// TIA Portal V20 export
// export: Created 2025-12-01T14:57:39.8501249Z, ExportSetting None, DisplayName Totally Integrated Automation Portal, DisplayVersion V20 Update 3, DisplayName TIA Portal Openness, DisplayVersion V20 Update 3, DisplayName TIA Portal Version Control Interface, DisplayVersion V20 Update 3, DisplayName STEP 7 Professional, DisplayVersion V20 Update 3, DisplayName STEP 7 Safety, DisplayVersion V20 Update 2, DisplayName WinCC Basic/Comfort/Advanced, DisplayVersion V20 Update 3, DisplayName WinCC Professional, DisplayVersion V20 Update 3, DisplayName WinCC Unified, DisplayVersion V20 Update 3
FUNCTION_BLOCK "FB371_DesApiladorDeCajasPlastico"   // FB371, LAD
TITLE = DesApilador de Cajas de Plastico
{ S7_Optimized_Access := 'FALSE' }
AUTHOR : MAQUINA
NAME : 20160211
VERSION : 3.2
// Dani Palacios: Modificación octubre 2017 para poder desabilitar la maquina con un bit (por ejemplo en la puesta a punto si no esta montada o en el simulador)
// La modificación esta sin probar y es todo lo relativo a la variable MaquinaDesHabilitada
// (bloqueo evolución desde etapa 0, bloqueo activación salidas en etapa 0 , fin vi sin mirar detectores y activación posición de reposo sin mirar detectores y variabkles de fin de movimiento).
// ES RESPONSABILIDAD DEL QUE DESABILITA LA MAQUINA QUE ESTA ESTE EN UNA POSICION QUE PERMITA EL MOVIMIENTO DE LAS CARGAS A TRAVES DE ELLA
// stored: AutoNumber false, SetENOAutomatically false
   VAR_INPUT
      Maquina : UInt;   // Numero de Maquina (Mesa)
      Error_Tx : Bool;   // Error en el Tx
      EnTension : Bool;   // Existe Tension en la Mesa
      NodoNoPresente : Bool;   // Nodo No Presente >>> Var. LENZE de Elevacion
      ByteInicial : Int;   // Byte Inicial >>> Var. LENZE de Elevacion
      MAQx_DesHabilitada : Bool;   // Config MAQ. >>> DesHabilitada
      MAQx_SinCentrador : Bool;   // Config MAQ. >>> No Activar Centrador
      MAQx_ActivarEspera : Bool;   // Config MAQ. >>> Sin Espera en Etapas
      TermicoFreno_ELEV : Bool;   // Termico del Freno de la Elevacion
      pHsMx_PresCarga : Bool;   // pHs de Presencia de Carga en la Maquina
      pHsMx_1 : Bool;   // pHs de la Mesa - Pos 1 de Av
      pHsMx_2 : Bool;   // pHs de la Mesa - Pos 2 de Av
      pHsMx_CrtSalida : Bool;   // pHs Control de Salida de Seguridad
      pHs_Referencia : Bool;   // pHs de Referencia >>> Var. LENZE de Elevacion
      EM_Up : Bool;   // Emergencia Arriba >>> Var. LENZE de Elevacion
      EM_Down : Bool;   // Emergencia Abajo >>> Var. LENZE de Elevacion
      CF1CF2_Cerrado : Bool;   // Centradores 1 y 2 Cerrados
      CF3CF4_Cerrado : Bool;   // Centradores 3 y 4 Cerrados
      CF5CF6_Cerrado : Bool;   // Centradores 5 y 6 Cerrados
      CF1CF2_Abierto : Bool;   // Centradores 1 y 2 Abiertos
      CF3CF4_Abierto : Bool;   // Centradores 3 y 4 Abiertos
      CF5CF6_Abierto : Bool;   // Centradores 5 y 6 Abiertos
      CM1CM2_Cerrado : Bool;   // Garras 1 y 2 Cerradas
      CM3CM4_Cerrado : Bool;   // Garras 3 y 4 Cerradas
      CM5CM6_Cerrado : Bool;   // Garras 5 y 6 Cerradas
      CM7CM8_Cerrado : Bool;   // Garras 7 y 8 Cerradas
      CM9CM10_Cerrado : Bool;   // Garras 9 y 10 Cerradas
      CM1CM2_Abierto : Bool;   // Garras 1 y 2 Abiertas
      CM3CM4_Abierto : Bool;   // Garras 3 y 4 Abiertas
      CM5CM6_Abierto : Bool;   // Garras 5 y 6 Abiertas
      CM7CM8_Abierto : Bool;   // Garras 7 y 8 Abiertas
      CM9CM10_Abierto : Bool;   // Garras 9 y 10 Abiertas
      GF1GF2_Cerrado : Bool;   // Guias superiores 1 y 2 Cerradas
      GF3GF4_Cerrado : Bool;   // Guias superiores 3 y 4 Cerradas
      GF1GF2_Abierto : Bool;   // Guias superiores 1 y 2 Abiertas
      GF3GF4_Abierto : Bool;   // Guias superiores 3 y 4 Abiertas
      EnMov_Centradores : Bool;   // Centradores >>> En Movimiento
      EnMov_Garras : Bool;   // Garras >>> En Movimiento
      EnMov_Guias : Bool;   // Guias >>> En Movimiento
      SubirManual : Bool;   // Subir en Manual >>> Var. LENZE de Elevacion
      BajarManual : Bool;   // Bajar en Manual >>> Var. LENZE de Elevacion
      AutoManual : Bool;   // Posicionar en Manual (Para realizar Test de Posicion)
      Homing : Bool;   // Homing >>> Var. LENZE de Elevacion
      DesApilador_FinSalida : Bool;   // Fin Salida >>> Interlock Mesa
      ActivarGuias : Bool;   // Activar las Guias Superiores (Por altura de la Pila)
      V_TOut_MovVertical : Int := 15000;   // TimeOut del Movimiento Vertical
      V_TOut_Centradores : Int := 5000;   // TimeOut de los Centradores
      V_TOut_Garras : Int := 5000;   // TimeOut de las Garras
      V_TOut_Guias : Int := 5000;   // TimeOut de las Guias Superiores
   END_VAR
   VAR_OUTPUT
      DesApilador_EnReposo : Bool;   // En Reposo >>> Interlock Maquina
      DesApilador_PermisoSalida : Bool;   // Permiso de Salida >>> Interlock Maquina
   END_VAR
   VAR
      PosicionActual : Int;   // Var. LENZE de Elevacion >>> Posicion Actual
      ErrorSubjet : Word;   // Var LENZE de Elevacion
      ErrorID : Word;   // Var LENZE de Elevacion
      PosicionManual : UInt;   // Posicion para el Test Manual
      PosicionInicial : UInt;   // TRACKING >>> Posicion Inicial de la Orden de DesApilar Cajas
      PosicionFinal : UInt;   // TRACKING >>> Posicion Final de la Orden de DesApilar Cajas
      TipoAmarre : UInt;   // TRACKING >>> Tipo de Amarre de las Garras de la Orden de DesApilar Cajas
      OrdenDesApilar : Bool;   // TRACKING >>> Orden de DesApilar Cajas
      Fin_OrdenDesApilar : Bool;   // TRACKING >>> Fin de la Orden de DesApilar Cajas
      Caja_TipoEuroPool : Bool;   // TRACKING >>> Caja de tipo EuroPool
      Caja_DosPequenas : Bool;   // TRACKING >>> La Fila es de Dos Cajas Pequeñas
      Caja_UnaPequena : Bool;   // TRACKING >>> La Fila es de Una Caja Pequeña
      Caja_Grande : Bool;   // TRACKING >>> La Fila es de Una Caja Grande
      EnPila_UnicaFila : Bool;   // TRACKING >>> La Pila es de Una Unica Fila
      Reset_ET00 : Bool;
      Reset_ET01 : Bool;
      DesApil_ET00 : Bool;
      DesApil_ET01 : Bool;
      DesApil_ET02 : Bool;
      DesApil_ET03 : Bool;
      DesApil_ET04 : Bool;
      DesApil_ET05 : Bool;
      DesApil_ET06 : Bool;
      DesApil_ET07 : Bool;
      DesApil_ET08 : Bool;
      PosicionIntermedia : UInt;   // AUXILIAR >>> Posicion Internedia de la Orden a Mover el Elevacion
      Posicion_OrdenMover : UInt;   // AUXILIAR >>> Posicion de la Orden a Mover el Elevacion
      OrdenMover : Bool;   // AUXILIAR >>> Orden de Mover el Elevacion
      Fin_OrdenMover : Bool;   // AUXILIAR >>> Orden de Mover el Elevacion
      MemoPosicionOK : Bool;   // AUXILIAR >>> Memoria de Posicion OK
      Carga_PosicionInicial : Bool;   // CARGA >>> Posicion Incial del DesApilado de Cajas
      Carga_PosicionIntermedia : Bool;   // CARGA >>> Posicion Intermedia del DesApilado de Cajas
      Carga_PosicionFinal : Bool;   // CARGA >>> Posicion Final del DesApilado de Cajas
      Carga_PosicionManual : Bool;   // CARGA >>> Posicion Manual de la Orden de Test
      ErrorVariador : Bool;   // AUXILIAR >>> Error del Variador
      ReferenciaOK : Bool;   // AUXILIAR >>> Referencia OK del Variador
      MemoHomingAuto : Bool;   // AUXILIAR >>> Memoria del Homing Automatico del Variador
      TIM_EsperaMover { S7_SetPoint := 'True'} : TON_TIME;   // TIM de Espera de Activar Orden al Var de LENZE (200ms)
      TIM_EsperaET02 { S7_SetPoint := 'True'} : TON_TIME;   // TIM de Espera para Activar ET02 (100ms)
      TIM_EsperaET04 { S7_SetPoint := 'True'} : TON_TIME;   // TIM de Espera para Activar ET04 (100ms)
      TMP_EnTension { S7_SetPoint := 'True'} : "FB910_CNT_UHS";
      TOut_MovVertical { S7_SetPoint := 'True'} : "FB910_CNT_UHS";   // TimeOut del Movimiento Vertical
      TOut_Centradores { S7_SetPoint := 'True'} : "FB910_CNT_UHS";   // TimeOut de los Centradores
      TOut_Garras { S7_SetPoint := 'True'} : "FB910_CNT_UHS";   // TimeOut de las Garras
      TOut_Guias { S7_SetPoint := 'True'} : "FB910_CNT_UHS";   // TimeOut de las Guias Superiores
      MA_Cerrar_CF1CF2 : Bool;   // ???
      MA_Cerrar_CF3CF4 : Bool;   // ???
      MA_Cerrar_CF5CF6 : Bool;   // ???
      MA_Abrir_CF1CF2 : Bool;   // ???
      MA_Abrir_CF3CF4 : Bool;   // ???
      MA_Abrir_CF5CF6 : Bool;   // ???
      MA_Cerrar_CM1CM2 : Bool;   // ???
      MA_Cerrar_CM3CM4 : Bool;   // ???
      MA_Cerrar_CM5CM6 : Bool;   // ???
      MA_Cerrar_CM7CM8 : Bool;   // ???
      MA_Cerrar_CM9CM10 : Bool;   // ???
      MA_Abrir_CM1CM2 : Bool;   // ???
      MA_Abrir_CM3CM4 : Bool;   // ???
      MA_Abrir_CM5CM6 : Bool;   // ???
      MA_Abrir_CM7CM8 : Bool;   // ???
      MA_Abrir_CM9CM10 : Bool;   // ???
      MA_Cerrar_GF1GF2 : Bool;   // ???
      MA_Cerrar_GF3GF4 : Bool;   // ???
      MA_Abrir_GF1GF2 : Bool;   // ???
      MA_Abrir_GF3GF4 : Bool;   // ???
   END_VAR
   VAR_TEMP
      EstadoZona : "EstadoZona";   // Estado de Zona de la Mesa
      EstadoMAQ : "EstadoMaquina_DesApiladorDeCajasPlastico";   // Estado del Vehiculo Inteliguente de la Maquina
      MAQx_AutoHoming : Bool;   // Config >>> Var. LENZE con Auto Homing
      MAQx_EncoderIncremental : Bool;   // Config >>> Var. LENZE con Encoder Incremental
      MAQx_ActivarAutoManual : Bool;   // Config >>> Activacion para el Test de posicionamiento manual
      CentradoresCerrados : Bool;   // AUXILIAR >>> Cerrados los Centradores
      CentradoresAbiertos : Bool;   // AUXILIAR >>> Abiertos los Centradores
      GarrasCerradas : Bool;   // AUXILIAR >>> Cerradas las Garras
      GarrasAbiertas : Bool;   // AUXILIAR >>> Abiertas las Garras
      GuiasCerradas : Bool;   // AUXILIAR >>> Cerradas las Guias Superiores
      GuiasAbiertas : Bool;   // AUXILIAR >>> Abiertas las Guias Superiores
      MA_CerrarCentradores : Bool;   // AUXILIAR >>> Cerrar los Centradores
      MA_AbrirCentradores : Bool;   // AUXILIAR >>> Abrir los Centradores
      MA_CerrarGarras : Bool;   // AUXILIAR >>> Cerrar las Garras
      MA_AbrirGarras : Bool;   // AUXILIAR >>> Abrir las Garras
      MA_CerrarGuias : Bool;   // AUXILIAR >>> Cerrar las Guias Superiores
      MA_AbrirGuias : Bool;   // AUXILIAR >>> Abrir las Guias Superiores
      AuxEstados : Bool;
   END_VAR
BEGIN

REGION Network 1: Configuraciones Especiales - Config >>> Var. LENZE de Elevacion
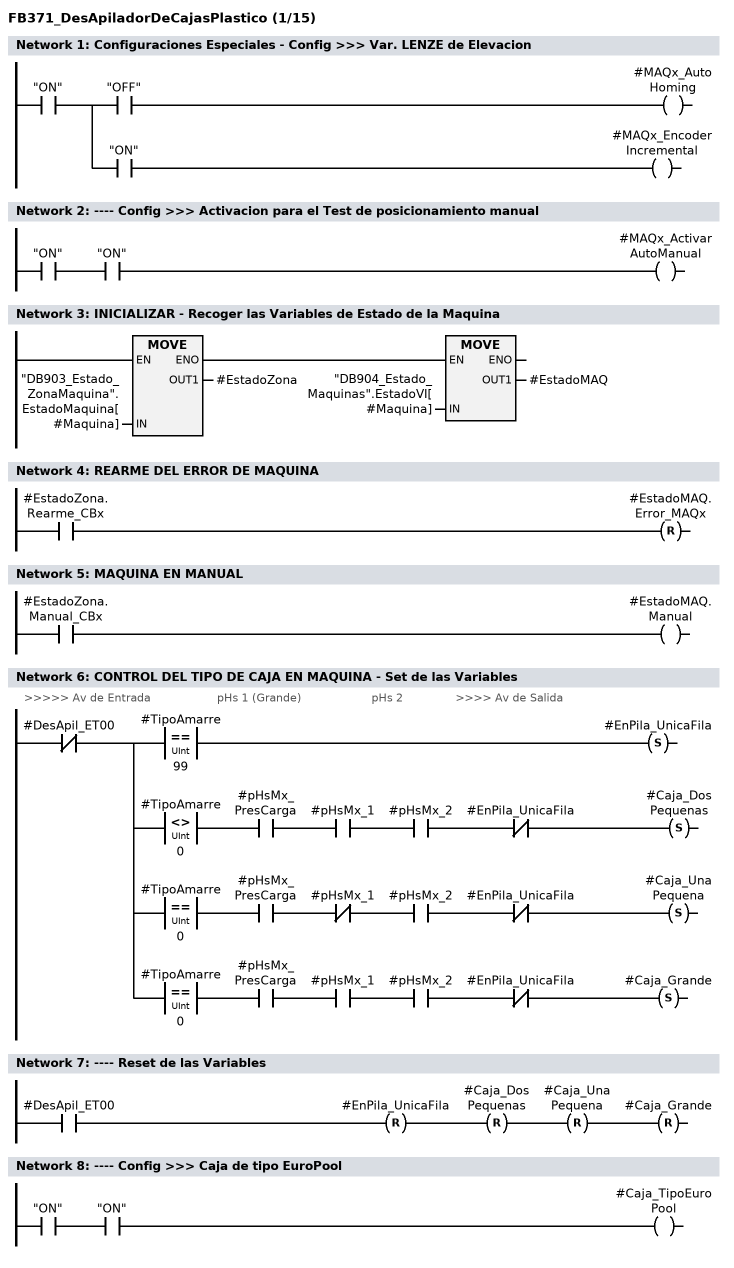
   RUNG wire#powerrail
      Contact( "ON" )
      wire#w1
      Contact( "OFF" )
      Coil( #MAQx_AutoHoming )
   END_RUNG
   RUNG wire#w1
      Contact( "ON" )
      Coil( #MAQx_EncoderIncremental )
   END_RUNG
   // the same network as SCL:
   #MAQx_AutoHoming := "ON" AND "OFF";
   #MAQx_EncoderIncremental := "ON" AND "ON";
END_REGION

REGION Network 2: ---- Config >>> Activacion para el Test de posicionamiento manual
   RUNG wire#powerrail
      Contact( "ON" )
      Contact( "ON" )
      Coil( #MAQx_ActivarAutoManual )
   END_RUNG
   // the same network as SCL:
   #MAQx_ActivarAutoManual := "ON" AND "ON";
END_REGION

REGION Network 3: INICIALIZAR - Recoger las Variables de Estado de la Maquina
   RUNG wire#powerrail
      Move(in := "DB903_Estado_ZonaMaquina".EstadoMaquina[#Maquina], out1 => #EstadoZona)
      Move(in := "DB904_Estado_Maquinas".EstadoVI[#Maquina], out1 => #EstadoMAQ)
   END_RUNG
   // the same network as SCL:
   #EstadoZona := "DB903_Estado_ZonaMaquina".EstadoMaquina[#Maquina];
   #EstadoMAQ := "DB904_Estado_Maquinas".EstadoVI[#Maquina];
END_REGION

REGION Network 4: REARME DEL ERROR DE MAQUINA
   RUNG wire#powerrail
      Contact( #EstadoZona.Rearme_CBx )
      R_Coil( #EstadoMAQ.Error_MAQx )
   END_RUNG
   // the same network as SCL:
   IF #EstadoZona.Rearme_CBx THEN #EstadoMAQ.Error_MAQx := FALSE; END_IF;
END_REGION

REGION Network 5: MAQUINA EN MANUAL
   RUNG wire#powerrail
      Contact( #EstadoZona.Manual_CBx )
      Coil( #EstadoMAQ.Manual )
   END_RUNG
   // the same network as SCL:
   #EstadoMAQ.Manual := #EstadoZona.Manual_CBx;
END_REGION

REGION Network 6: CONTROL DEL TIPO DE CAJA EN MAQUINA - Set de las Variables
   // >>>>> Av de Entrada                   pHs 1 (Grande)                    pHs 2               >>>> Av de Salida
   RUNG wire#powerrail
      I_Contact( #DesApil_ET00 )
      wire#w1
      { S7_Templates := "SrcType := UInt" } EQ_Contact(in1 := #TipoAmarre, in2 := 99)
      S_Coil( #EnPila_UnicaFila )
   END_RUNG
   RUNG wire#w1
      { S7_Templates := "SrcType := UInt" } NE_Contact(in1 := #TipoAmarre, in2 := 0)
      Contact( #pHsMx_PresCarga )
      Contact( #pHsMx_1 )
      Contact( #pHsMx_2 )
      I_Contact( #EnPila_UnicaFila )
      S_Coil( #Caja_DosPequenas )
   END_RUNG
   RUNG wire#w1
      { S7_Templates := "SrcType := UInt" } EQ_Contact(in1 := #TipoAmarre, in2 := 0)
      Contact( #pHsMx_PresCarga )
      I_Contact( #pHsMx_1 )
      Contact( #pHsMx_2 )
      I_Contact( #EnPila_UnicaFila )
      S_Coil( #Caja_UnaPequena )
   END_RUNG
   RUNG wire#w1
      { S7_Templates := "SrcType := UInt" } EQ_Contact(in1 := #TipoAmarre, in2 := 0)
      Contact( #pHsMx_PresCarga )
      Contact( #pHsMx_1 )
      Contact( #pHsMx_2 )
      I_Contact( #EnPila_UnicaFila )
      S_Coil( #Caja_Grande )
   END_RUNG
   // the same network as SCL:
   IF NOT #DesApil_ET00 AND (#TipoAmarre = 99) THEN #EnPila_UnicaFila := TRUE; END_IF;
   IF NOT #DesApil_ET00 AND (#TipoAmarre <> 0) AND #pHsMx_PresCarga AND #pHsMx_1 AND #pHsMx_2 AND NOT #EnPila_UnicaFila THEN
       #Caja_DosPequenas := TRUE;
   END_IF;
   IF NOT #DesApil_ET00 AND (#TipoAmarre = 0) AND #pHsMx_PresCarga AND NOT #pHsMx_1 AND #pHsMx_2 AND NOT #EnPila_UnicaFila THEN
       #Caja_UnaPequena := TRUE;
   END_IF;
   IF NOT #DesApil_ET00 AND (#TipoAmarre = 0) AND #pHsMx_PresCarga AND #pHsMx_1 AND #pHsMx_2 AND NOT #EnPila_UnicaFila THEN
       #Caja_Grande := TRUE;
   END_IF;
END_REGION

REGION Network 7: ---- Reset de las Variables
   RUNG wire#powerrail
      Contact( #DesApil_ET00 )
      R_Coil( #EnPila_UnicaFila )
      R_Coil( #Caja_DosPequenas )
      R_Coil( #Caja_UnaPequena )
      R_Coil( #Caja_Grande )
   END_RUNG
   // the same network as SCL:
   IF #DesApil_ET00 THEN
       #EnPila_UnicaFila := FALSE;
       #Caja_DosPequenas := FALSE;
       #Caja_UnaPequena := FALSE;
       #Caja_Grande := FALSE;
   END_IF;
END_REGION

REGION Network 8: ---- Config >>> Caja de tipo EuroPool
   RUNG wire#powerrail
      Contact( "ON" )
      Contact( "ON" )
      Coil( #Caja_TipoEuroPool )
   END_RUNG
   // the same network as SCL:
   #Caja_TipoEuroPool := "ON" AND "ON";
END_REGION

REGION Network 9: VARIABLES AUXILIARES - Control de Centradores - Cerrados
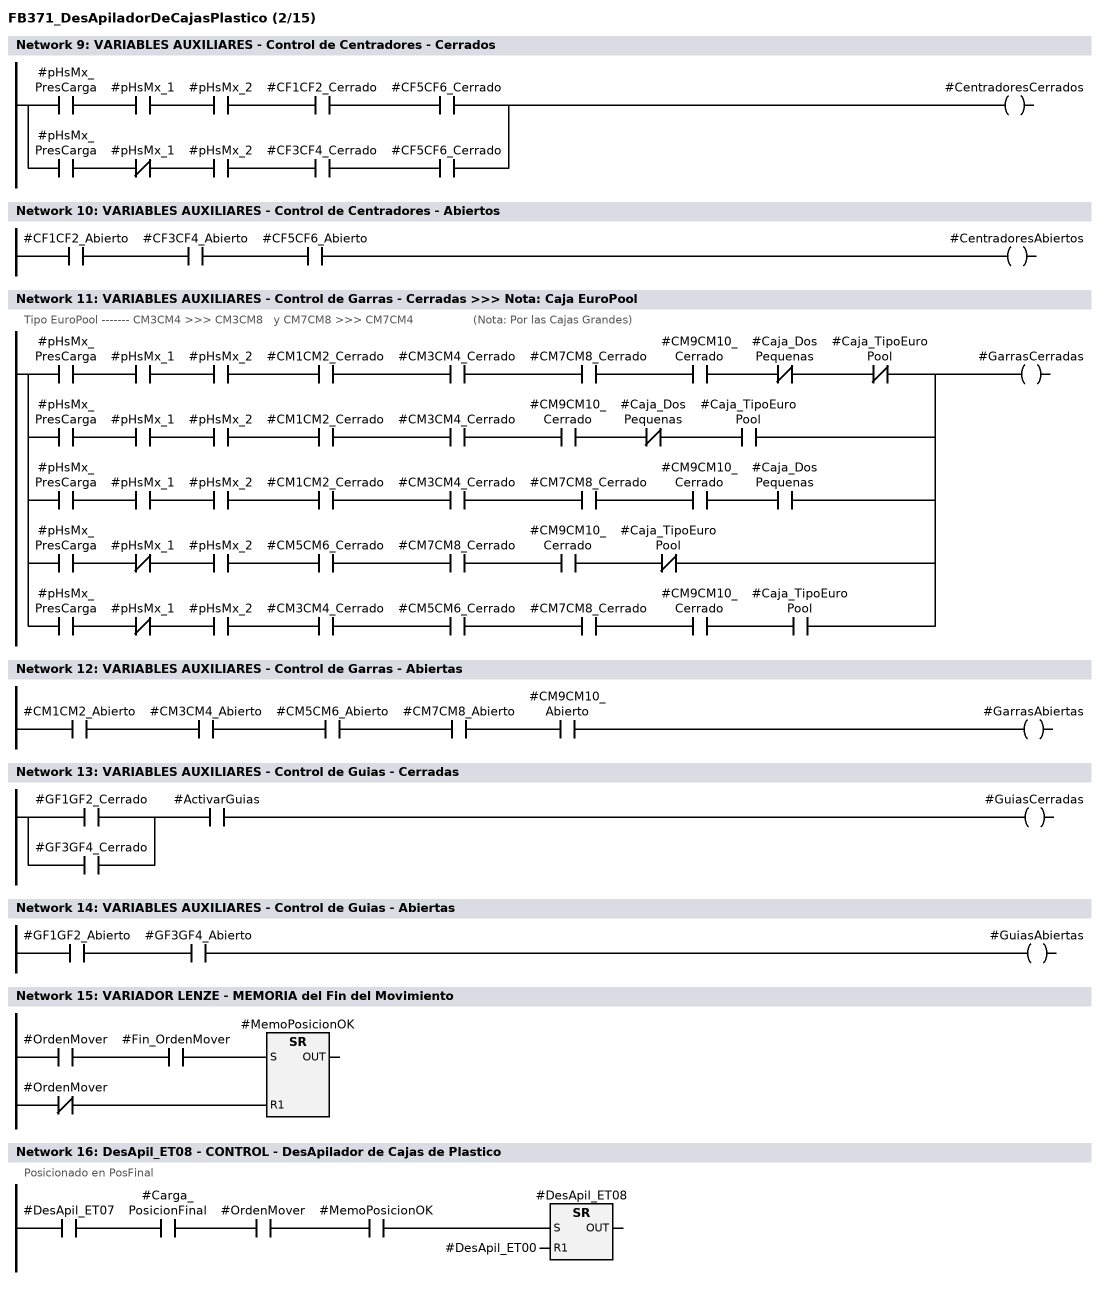
   RUNG wire#powerrail
      Contact( #pHsMx_PresCarga )
      Contact( #pHsMx_1 )
      Contact( #pHsMx_2 )
      Contact( #CF1CF2_Cerrado )
      Contact( #CF5CF6_Cerrado )
      wire#w1
      Coil( #CentradoresCerrados )
   END_RUNG
   RUNG wire#powerrail
      Contact( #pHsMx_PresCarga )
      I_Contact( #pHsMx_1 )
      Contact( #pHsMx_2 )
      Contact( #CF3CF4_Cerrado )
      Contact( #CF5CF6_Cerrado )
   END_RUNG wire#w1
   // the same network as SCL:
   #CentradoresCerrados := (#pHsMx_PresCarga AND #pHsMx_1 AND #pHsMx_2 AND #CF1CF2_Cerrado AND #CF5CF6_Cerrado) OR (#pHsMx_PresCarga AND NOT #pHsMx_1 AND #pHsMx_2 AND #CF3CF4_Cerrado AND #CF5CF6_Cerrado);
END_REGION

REGION Network 10: VARIABLES AUXILIARES - Control de Centradores - Abiertos
   RUNG wire#powerrail
      Contact( #CF1CF2_Abierto )
      Contact( #CF3CF4_Abierto )
      Contact( #CF5CF6_Abierto )
      Coil( #CentradoresAbiertos )
   END_RUNG
   // the same network as SCL:
   #CentradoresAbiertos := #CF1CF2_Abierto AND #CF3CF4_Abierto AND #CF5CF6_Abierto;
END_REGION

REGION Network 11: VARIABLES AUXILIARES - Control de Garras - Cerradas >>> Nota: Caja EuroPool
   // Tipo EuroPool ------- CM3CM4 >>> CM3CM8   y CM7CM8 >>> CM7CM4                 (Nota: Por las Cajas Grandes)
   RUNG wire#powerrail
      Contact( #pHsMx_PresCarga )
      Contact( #pHsMx_1 )
      Contact( #pHsMx_2 )
      Contact( #CM1CM2_Cerrado )
      Contact( #CM3CM4_Cerrado )
      Contact( #CM7CM8_Cerrado )
      Contact( #CM9CM10_Cerrado )
      I_Contact( #Caja_DosPequenas )
      I_Contact( #Caja_TipoEuroPool )
      wire#w1
      Coil( #GarrasCerradas )
   END_RUNG
   RUNG wire#powerrail
      Contact( #pHsMx_PresCarga )
      Contact( #pHsMx_1 )
      Contact( #pHsMx_2 )
      Contact( #CM1CM2_Cerrado )
      Contact( #CM3CM4_Cerrado )
      Contact( #CM9CM10_Cerrado )
      I_Contact( #Caja_DosPequenas )
      Contact( #Caja_TipoEuroPool )
   END_RUNG wire#w1
   RUNG wire#powerrail
      Contact( #pHsMx_PresCarga )
      Contact( #pHsMx_1 )
      Contact( #pHsMx_2 )
      Contact( #CM1CM2_Cerrado )
      Contact( #CM3CM4_Cerrado )
      Contact( #CM7CM8_Cerrado )
      Contact( #CM9CM10_Cerrado )
      Contact( #Caja_DosPequenas )
   END_RUNG wire#w1
   RUNG wire#powerrail
      Contact( #pHsMx_PresCarga )
      I_Contact( #pHsMx_1 )
      Contact( #pHsMx_2 )
      Contact( #CM5CM6_Cerrado )
      Contact( #CM7CM8_Cerrado )
      Contact( #CM9CM10_Cerrado )
      I_Contact( #Caja_TipoEuroPool )
   END_RUNG wire#w1
   RUNG wire#powerrail
      Contact( #pHsMx_PresCarga )
      I_Contact( #pHsMx_1 )
      Contact( #pHsMx_2 )
      Contact( #CM3CM4_Cerrado )
      Contact( #CM5CM6_Cerrado )
      Contact( #CM7CM8_Cerrado )
      Contact( #CM9CM10_Cerrado )
      Contact( #Caja_TipoEuroPool )
   END_RUNG wire#w1
   // the same network as SCL:
   #GarrasCerradas := (#pHsMx_PresCarga AND #pHsMx_1 AND #pHsMx_2 AND #CM1CM2_Cerrado AND #CM3CM4_Cerrado AND #CM7CM8_Cerrado AND #CM9CM10_Cerrado AND NOT #Caja_DosPequenas AND NOT #Caja_TipoEuroPool) OR (#pHsMx_PresCarga AND #pHsMx_1 AND #pHsMx_2 AND #CM1CM2_Cerrado AND #CM3CM4_Cerrado AND #CM9CM10_Cerrado AND NOT #Caja_DosPequenas AND #Caja_TipoEuroPool) OR (#pHsMx_PresCarga AND #pHsMx_1 AND #pHsMx_2 AND #CM1CM2_Cerrado AND #CM3CM4_Cerrado AND #CM7CM8_Cerrado AND #CM9CM10_Cerrado AND #Caja_DosPequenas) OR (#pHsMx_PresCarga AND NOT #pHsMx_1 AND #pHsMx_2 AND #CM5CM6_Cerrado AND #CM7CM8_Cerrado AND #CM9CM10_Cerrado AND NOT #Caja_TipoEuroPool) OR (#pHsMx_PresCarga AND NOT #pHsMx_1 AND #pHsMx_2 AND #CM3CM4_Cerrado AND #CM5CM6_Cerrado AND #CM7CM8_Cerrado AND #CM9CM10_Cerrado AND #Caja_TipoEuroPool);
END_REGION

REGION Network 12: VARIABLES AUXILIARES - Control de Garras - Abiertas
   RUNG wire#powerrail
      Contact( #CM1CM2_Abierto )
      Contact( #CM3CM4_Abierto )
      Contact( #CM5CM6_Abierto )
      Contact( #CM7CM8_Abierto )
      Contact( #CM9CM10_Abierto )
      Coil( #GarrasAbiertas )
   END_RUNG
   // the same network as SCL:
   #GarrasAbiertas := #CM1CM2_Abierto AND #CM3CM4_Abierto AND #CM5CM6_Abierto AND #CM7CM8_Abierto AND #CM9CM10_Abierto;
END_REGION

REGION Network 13: VARIABLES AUXILIARES - Control de Guias - Cerradas
   RUNG wire#powerrail
      Contact( #GF1GF2_Cerrado )
      wire#w1
      Contact( #ActivarGuias )
      Coil( #GuiasCerradas )
   END_RUNG
   RUNG wire#powerrail
      Contact( #GF3GF4_Cerrado )
   END_RUNG wire#w1
   // the same network as SCL:
   #GuiasCerradas := (#GF1GF2_Cerrado OR #GF3GF4_Cerrado) AND #ActivarGuias;
END_REGION

REGION Network 14: VARIABLES AUXILIARES - Control de Guias - Abiertas
   RUNG wire#powerrail
      Contact( #GF1GF2_Abierto )
      Contact( #GF3GF4_Abierto )
      Coil( #GuiasAbiertas )
   END_RUNG
   // the same network as SCL:
   #GuiasAbiertas := #GF1GF2_Abierto AND #GF3GF4_Abierto;
END_REGION

REGION Network 15: VARIADOR LENZE - MEMORIA del Fin del Movimiento
   RUNG wire#powerrail
      Contact( #OrdenMover )
      Contact( #Fin_OrdenMover )
      S_SR(operand := #MemoPosicionOK, r1 := wire#w1)
   END_RUNG
   RUNG wire#powerrail
      I_Contact( #OrdenMover )
   END_RUNG wire#w1
   // the same network as SCL:
   IF #OrdenMover AND #Fin_OrdenMover THEN
       #MemoPosicionOK := TRUE;   // SR flip-flop
   END_IF;
   IF NOT #OrdenMover THEN #MemoPosicionOK := FALSE; END_IF;
END_REGION

REGION Network 16: DesApil_ET08 - CONTROL - DesApilador de Cajas de Plastico
   // Posicionado en PosFinal
   RUNG wire#powerrail
      Contact( #DesApil_ET07 )
      Contact( #Carga_PosicionFinal )
      Contact( #OrdenMover )
      Contact( #MemoPosicionOK )
      S_SR(operand := #DesApil_ET08, r1 := #DesApil_ET00)
   END_RUNG
   // the same network as SCL:
   IF #DesApil_ET07 AND #Carga_PosicionFinal AND #OrdenMover AND #MemoPosicionOK THEN
       #DesApil_ET08 := TRUE;   // SR flip-flop
   END_IF;
   IF #DesApil_ET00 THEN #DesApil_ET08 := FALSE; END_IF;
END_REGION

REGION Network 17: DesApil_ET07
   // A Salido la Caja
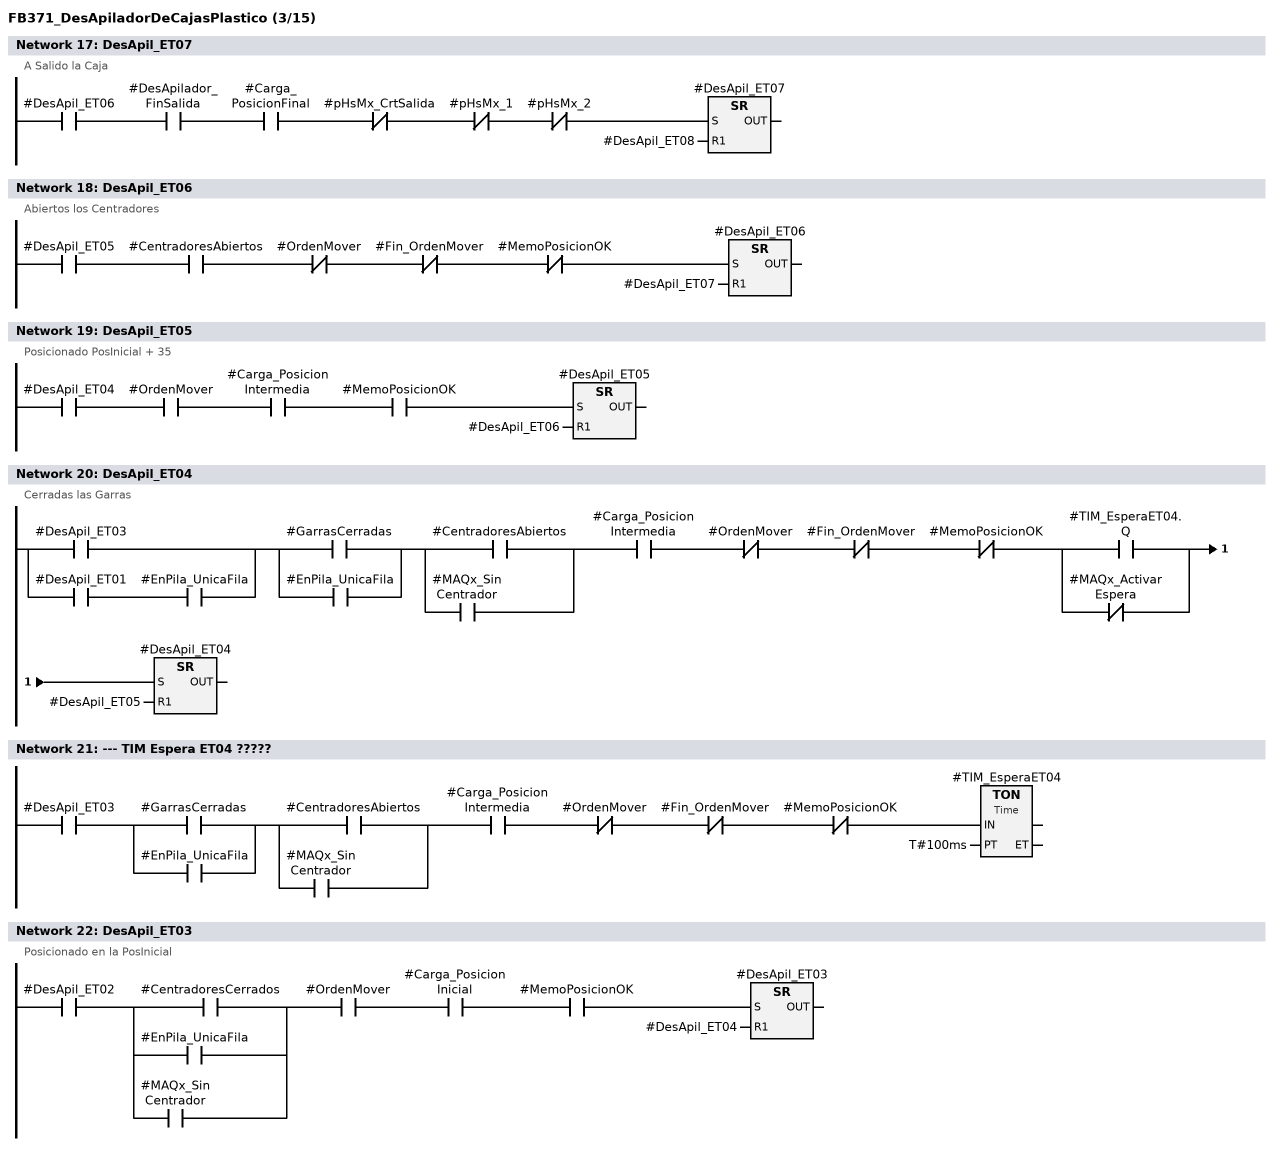
   RUNG wire#powerrail
      Contact( #DesApil_ET06 )
      Contact( #DesApilador_FinSalida )
      Contact( #Carga_PosicionFinal )
      I_Contact( #pHsMx_CrtSalida )
      I_Contact( #pHsMx_1 )
      I_Contact( #pHsMx_2 )
      S_SR(operand := #DesApil_ET07, r1 := #DesApil_ET08)
   END_RUNG
   // the same network as SCL:
   IF #DesApil_ET06 AND #DesApilador_FinSalida AND #Carga_PosicionFinal AND NOT #pHsMx_CrtSalida AND NOT #pHsMx_1 AND NOT #pHsMx_2 THEN
       #DesApil_ET07 := TRUE;   // SR flip-flop
   END_IF;
   IF #DesApil_ET08 THEN #DesApil_ET07 := FALSE; END_IF;
END_REGION

REGION Network 18: DesApil_ET06
   // Abiertos los Centradores
   RUNG wire#powerrail
      Contact( #DesApil_ET05 )
      Contact( #CentradoresAbiertos )
      I_Contact( #OrdenMover )
      I_Contact( #Fin_OrdenMover )
      I_Contact( #MemoPosicionOK )
      S_SR(operand := #DesApil_ET06, r1 := #DesApil_ET07)
   END_RUNG
   // the same network as SCL:
   IF #DesApil_ET05 AND #CentradoresAbiertos AND NOT #OrdenMover AND NOT #Fin_OrdenMover AND NOT #MemoPosicionOK THEN
       #DesApil_ET06 := TRUE;   // SR flip-flop
   END_IF;
   IF #DesApil_ET07 THEN #DesApil_ET06 := FALSE; END_IF;
END_REGION

REGION Network 19: DesApil_ET05
   // Posicionado PosInicial + 35
   RUNG wire#powerrail
      Contact( #DesApil_ET04 )
      Contact( #OrdenMover )
      Contact( #Carga_PosicionIntermedia )
      Contact( #MemoPosicionOK )
      S_SR(operand := #DesApil_ET05, r1 := #DesApil_ET06)
   END_RUNG
   // the same network as SCL:
   IF #DesApil_ET04 AND #OrdenMover AND #Carga_PosicionIntermedia AND #MemoPosicionOK THEN
       #DesApil_ET05 := TRUE;   // SR flip-flop
   END_IF;
   IF #DesApil_ET06 THEN #DesApil_ET05 := FALSE; END_IF;
END_REGION

REGION Network 20: DesApil_ET04
   // Cerradas las Garras
   RUNG wire#powerrail
      Contact( #DesApil_ET03 )
      wire#w1
      Contact( #GarrasCerradas )
      wire#w2
      Contact( #CentradoresAbiertos )
      wire#w3
      Contact( #Carga_PosicionIntermedia )
      I_Contact( #OrdenMover )
      I_Contact( #Fin_OrdenMover )
      I_Contact( #MemoPosicionOK )
      wire#w4
      Contact( #TIM_EsperaET04.Q )
      wire#w5
      S_SR(operand := #DesApil_ET04, r1 := #DesApil_ET05)
   END_RUNG
   RUNG wire#powerrail
      Contact( #DesApil_ET01 )
      Contact( #EnPila_UnicaFila )
   END_RUNG wire#w1
   RUNG wire#w1
      Contact( #EnPila_UnicaFila )
   END_RUNG wire#w2
   RUNG wire#w2
      Contact( #MAQx_SinCentrador )
   END_RUNG wire#w3
   RUNG wire#w4
      I_Contact( #MAQx_ActivarEspera )
   END_RUNG wire#w5
   // the same network as SCL:
   IF (#DesApil_ET03 OR (#DesApil_ET01 AND #EnPila_UnicaFila)) AND (#GarrasCerradas OR #EnPila_UnicaFila) AND (#CentradoresAbiertos OR #MAQx_SinCentrador) AND #Carga_PosicionIntermedia AND NOT #OrdenMover AND NOT #Fin_OrdenMover AND NOT #MemoPosicionOK AND (#TIM_EsperaET04.Q OR NOT #MAQx_ActivarEspera) THEN
       #DesApil_ET04 := TRUE;   // SR flip-flop
   END_IF;
   IF #DesApil_ET05 THEN #DesApil_ET04 := FALSE; END_IF;
END_REGION

REGION Network 21: --- TIM Espera ET04 ?????
   RUNG wire#powerrail
      Contact( #DesApil_ET03 )
      wire#w1
      Contact( #GarrasCerradas )
      wire#w2
      Contact( #CentradoresAbiertos )
      wire#w3
      Contact( #Carga_PosicionIntermedia )
      I_Contact( #OrdenMover )
      I_Contact( #Fin_OrdenMover )
      I_Contact( #MemoPosicionOK )
      { S7_Templates := "time_type := Time" } #TIM_EsperaET04.TON(pt := T#100ms, et =>)
   END_RUNG
   RUNG wire#w1
      Contact( #EnPila_UnicaFila )
   END_RUNG wire#w2
   RUNG wire#w2
      Contact( #MAQx_SinCentrador )
   END_RUNG wire#w3
   // the same network as SCL:
   #TIM_EsperaET04(IN := #DesApil_ET03 AND (#GarrasCerradas OR #EnPila_UnicaFila) AND (#CentradoresAbiertos OR #MAQx_SinCentrador) AND #Carga_PosicionIntermedia AND NOT #OrdenMover AND NOT #Fin_OrdenMover AND NOT #MemoPosicionOK,   // TON
                   PT := T#100ms);
END_REGION

REGION Network 22: DesApil_ET03
   // Posicionado en la PosInicial
   RUNG wire#powerrail
      Contact( #DesApil_ET02 )
      wire#w1
      Contact( #CentradoresCerrados )
      wire#w2
      Contact( #OrdenMover )
      Contact( #Carga_PosicionInicial )
      Contact( #MemoPosicionOK )
      S_SR(operand := #DesApil_ET03, r1 := #DesApil_ET04)
   END_RUNG
   RUNG wire#w1
      Contact( #EnPila_UnicaFila )
   END_RUNG wire#w2
   RUNG wire#w1
      Contact( #MAQx_SinCentrador )
   END_RUNG wire#w2
   // the same network as SCL:
   IF #DesApil_ET02 AND (#CentradoresCerrados OR #EnPila_UnicaFila OR #MAQx_SinCentrador) AND #OrdenMover AND #Carga_PosicionInicial AND #MemoPosicionOK THEN
       #DesApil_ET03 := TRUE;   // SR flip-flop
   END_IF;
   IF #DesApil_ET04 THEN #DesApil_ET03 := FALSE; END_IF;
END_REGION

REGION Network 23: DesApil_ET02
   // Cerrados los Centradores
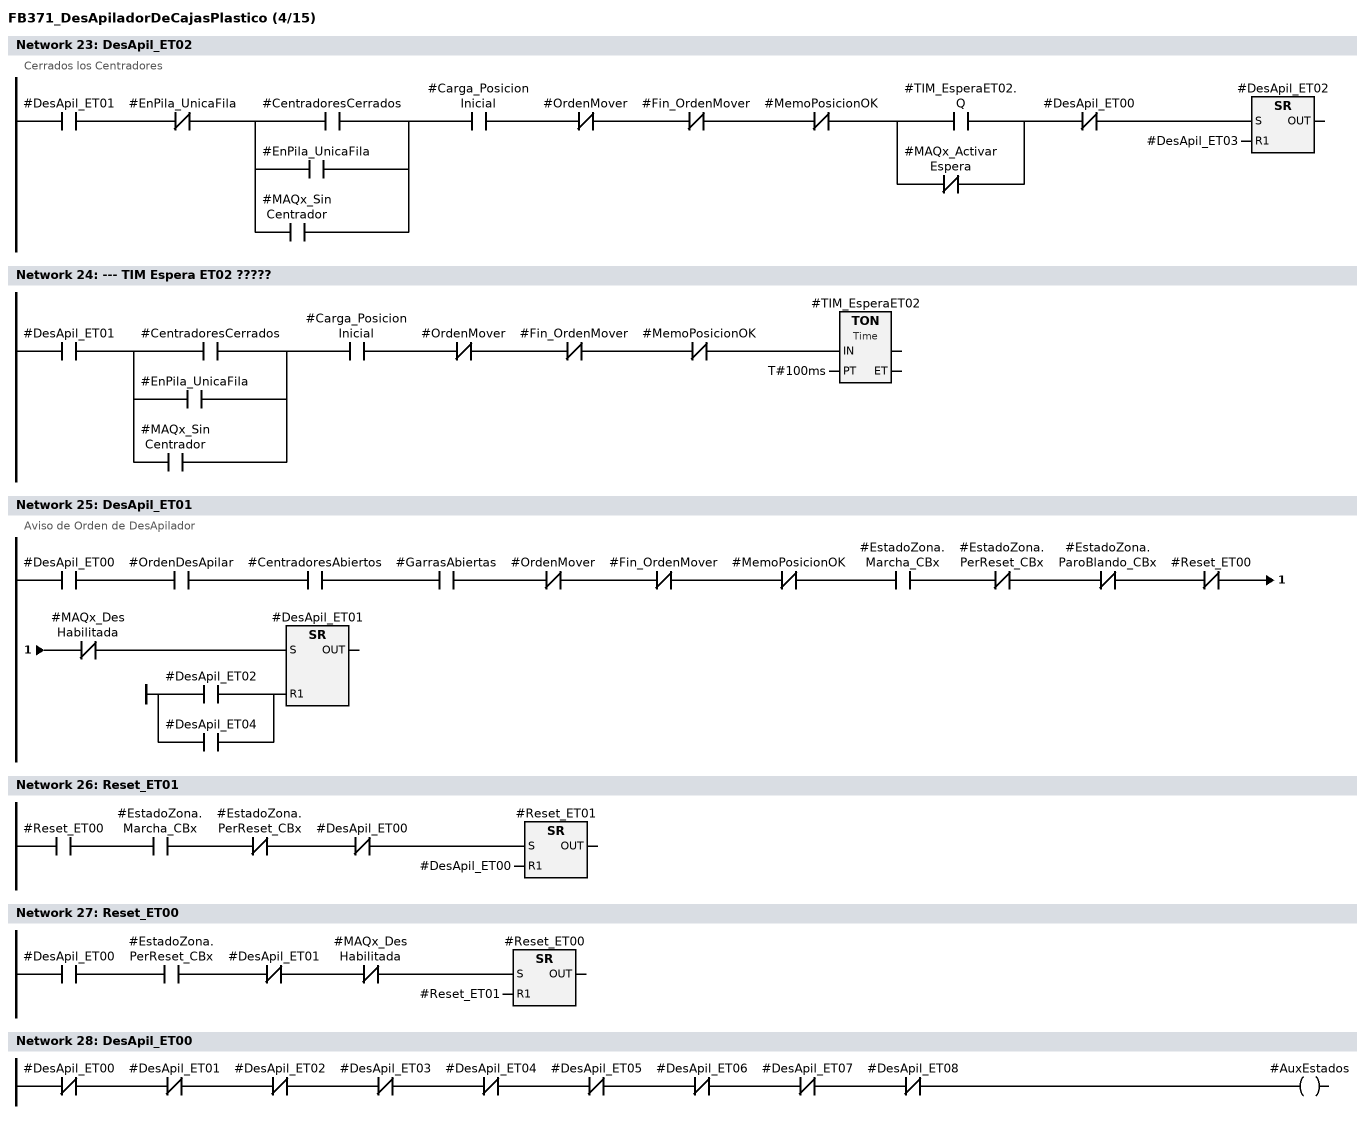
   RUNG wire#powerrail
      Contact( #DesApil_ET01 )
      I_Contact( #EnPila_UnicaFila )
      wire#w1
      Contact( #CentradoresCerrados )
      wire#w2
      Contact( #Carga_PosicionInicial )
      I_Contact( #OrdenMover )
      I_Contact( #Fin_OrdenMover )
      I_Contact( #MemoPosicionOK )
      wire#w3
      Contact( #TIM_EsperaET02.Q )
      wire#w4
      I_Contact( #DesApil_ET00 )
      S_SR(operand := #DesApil_ET02, r1 := #DesApil_ET03)
   END_RUNG
   RUNG wire#w1
      Contact( #EnPila_UnicaFila )
   END_RUNG wire#w2
   RUNG wire#w1
      Contact( #MAQx_SinCentrador )
   END_RUNG wire#w2
   RUNG wire#w3
      I_Contact( #MAQx_ActivarEspera )
   END_RUNG wire#w4
   // the same network as SCL:
   IF #DesApil_ET01 AND NOT #EnPila_UnicaFila AND (#CentradoresCerrados OR #EnPila_UnicaFila OR #MAQx_SinCentrador) AND #Carga_PosicionInicial AND NOT #OrdenMover AND NOT #Fin_OrdenMover AND NOT #MemoPosicionOK AND (#TIM_EsperaET02.Q OR NOT #MAQx_ActivarEspera) AND NOT #DesApil_ET00 THEN
       #DesApil_ET02 := TRUE;   // SR flip-flop
   END_IF;
   IF #DesApil_ET03 THEN #DesApil_ET02 := FALSE; END_IF;
END_REGION

REGION Network 24: --- TIM Espera ET02 ?????
   RUNG wire#powerrail
      Contact( #DesApil_ET01 )
      wire#w1
      Contact( #CentradoresCerrados )
      wire#w2
      Contact( #Carga_PosicionInicial )
      I_Contact( #OrdenMover )
      I_Contact( #Fin_OrdenMover )
      I_Contact( #MemoPosicionOK )
      { S7_Templates := "time_type := Time" } #TIM_EsperaET02.TON(pt := T#100ms, et =>)
   END_RUNG
   RUNG wire#w1
      Contact( #EnPila_UnicaFila )
   END_RUNG wire#w2
   RUNG wire#w1
      Contact( #MAQx_SinCentrador )
   END_RUNG wire#w2
   // the same network as SCL:
   #TIM_EsperaET02(IN := #DesApil_ET01 AND (#CentradoresCerrados OR #EnPila_UnicaFila OR #MAQx_SinCentrador) AND #Carga_PosicionInicial AND NOT #OrdenMover AND NOT #Fin_OrdenMover AND NOT #MemoPosicionOK,   // TON
                   PT := T#100ms);
END_REGION

REGION Network 25: DesApil_ET01
   // Aviso de Orden de DesApilador
   RUNG wire#powerrail
      Contact( #DesApil_ET00 )
      Contact( #OrdenDesApilar )
      Contact( #CentradoresAbiertos )
      Contact( #GarrasAbiertas )
      I_Contact( #OrdenMover )
      I_Contact( #Fin_OrdenMover )
      I_Contact( #MemoPosicionOK )
      Contact( #EstadoZona.Marcha_CBx )
      I_Contact( #EstadoZona.PerReset_CBx )
      I_Contact( #EstadoZona.ParoBlando_CBx )
      I_Contact( #Reset_ET00 )
      I_Contact( #MAQx_DesHabilitada )
      S_SR(operand := #DesApil_ET01, r1 := wire#w1)
   END_RUNG
   RUNG wire#powerrail
      Contact( #DesApil_ET02 )
   END_RUNG wire#w1
   RUNG wire#powerrail
      Contact( #DesApil_ET04 )
   END_RUNG wire#w1
   // the same network as SCL:
   IF #DesApil_ET00 AND #OrdenDesApilar AND #CentradoresAbiertos AND #GarrasAbiertas AND NOT #OrdenMover AND NOT #Fin_OrdenMover AND NOT #MemoPosicionOK AND #EstadoZona.Marcha_CBx AND NOT #EstadoZona.PerReset_CBx AND NOT #EstadoZona.ParoBlando_CBx AND NOT #Reset_ET00 AND NOT #MAQx_DesHabilitada THEN
       #DesApil_ET01 := TRUE;   // SR flip-flop
   END_IF;
   IF #DesApil_ET02 OR #DesApil_ET04 THEN #DesApil_ET01 := FALSE; END_IF;
END_REGION

REGION Network 26: Reset_ET01
   RUNG wire#powerrail
      Contact( #Reset_ET00 )
      Contact( #EstadoZona.Marcha_CBx )
      I_Contact( #EstadoZona.PerReset_CBx )
      I_Contact( #DesApil_ET00 )
      S_SR(operand := #Reset_ET01, r1 := #DesApil_ET00)
   END_RUNG
   // the same network as SCL:
   IF #Reset_ET00 AND #EstadoZona.Marcha_CBx AND NOT #EstadoZona.PerReset_CBx AND NOT #DesApil_ET00 THEN
       #Reset_ET01 := TRUE;   // SR flip-flop
   END_IF;
   IF #DesApil_ET00 THEN #Reset_ET01 := FALSE; END_IF;
END_REGION

REGION Network 27: Reset_ET00
   RUNG wire#powerrail
      Contact( #DesApil_ET00 )
      Contact( #EstadoZona.PerReset_CBx )
      I_Contact( #DesApil_ET01 )
      I_Contact( #MAQx_DesHabilitada )
      S_SR(operand := #Reset_ET00, r1 := #Reset_ET01)
   END_RUNG
   // the same network as SCL:
   IF #DesApil_ET00 AND #EstadoZona.PerReset_CBx AND NOT #DesApil_ET01 AND NOT #MAQx_DesHabilitada THEN
       #Reset_ET00 := TRUE;   // SR flip-flop
   END_IF;
   IF #Reset_ET01 THEN #Reset_ET00 := FALSE; END_IF;
END_REGION

REGION Network 28: DesApil_ET00
   RUNG wire#powerrail
      I_Contact( #DesApil_ET00 )
      I_Contact( #DesApil_ET01 )
      I_Contact( #DesApil_ET02 )
      I_Contact( #DesApil_ET03 )
      I_Contact( #DesApil_ET04 )
      I_Contact( #DesApil_ET05 )
      I_Contact( #DesApil_ET06 )
      I_Contact( #DesApil_ET07 )
      I_Contact( #DesApil_ET08 )
      Coil( #AuxEstados )
   END_RUNG
   // the same network as SCL:
   #AuxEstados := NOT #DesApil_ET00 AND NOT #DesApil_ET01 AND NOT #DesApil_ET02 AND NOT #DesApil_ET03 AND NOT #DesApil_ET04 AND NOT #DesApil_ET05 AND NOT #DesApil_ET06 AND NOT #DesApil_ET07 AND NOT #DesApil_ET08;
END_REGION

REGION Network 29: ---
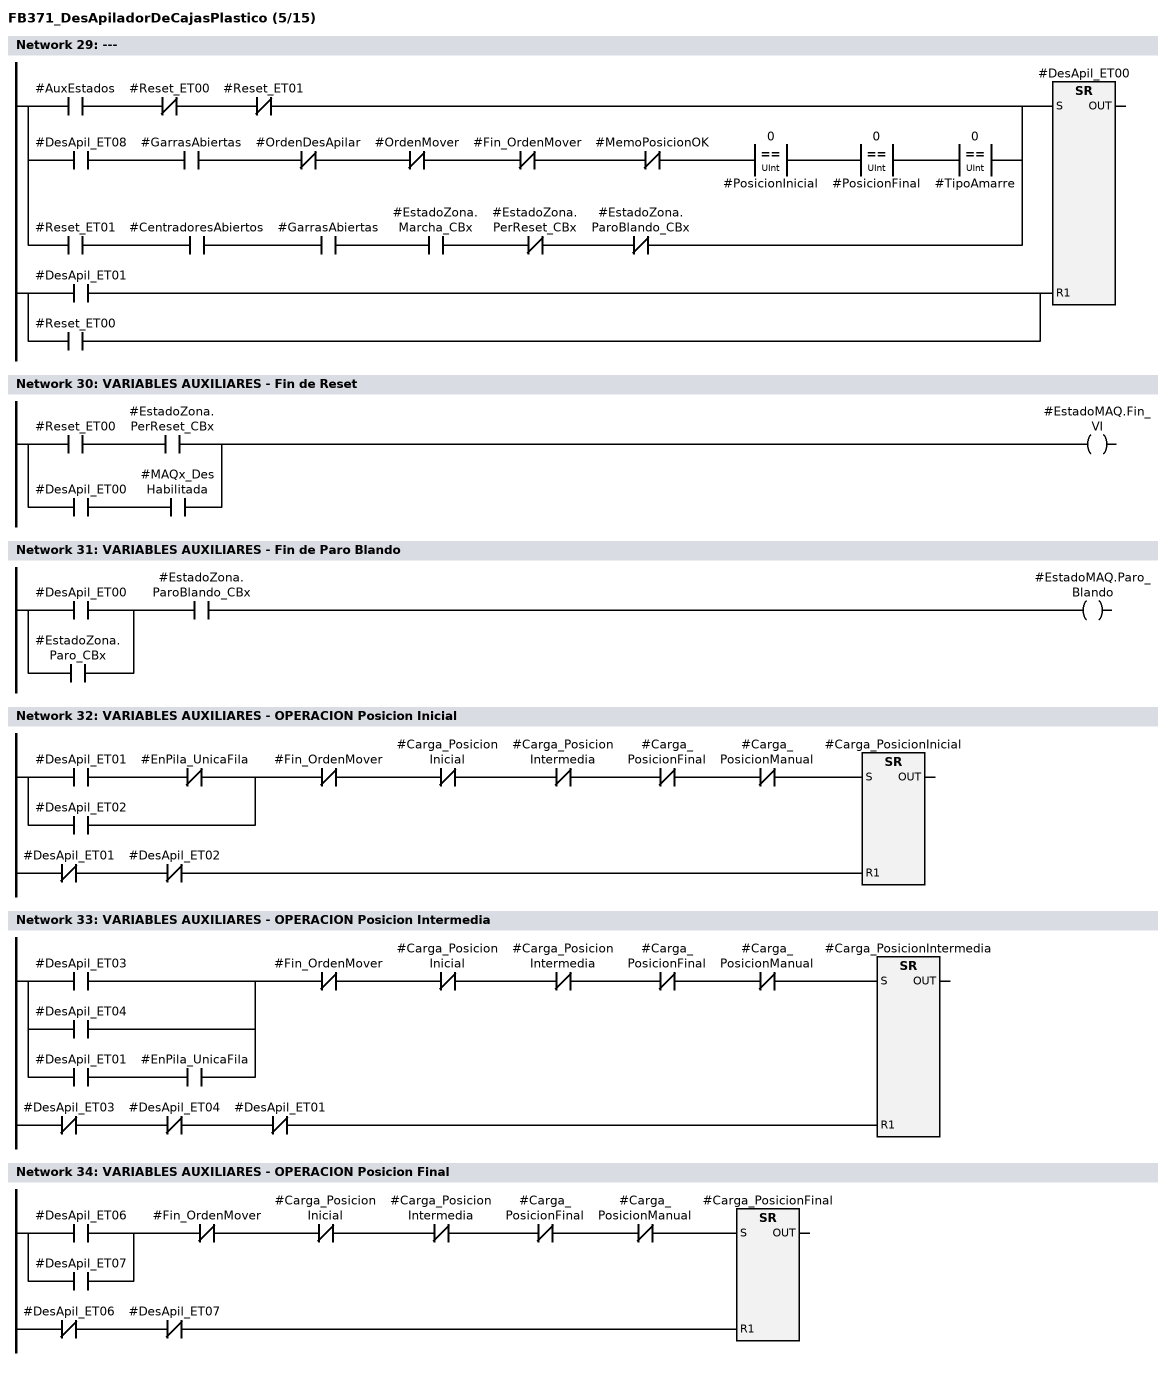
   RUNG wire#powerrail
      Contact( #AuxEstados )
      I_Contact( #Reset_ET00 )
      I_Contact( #Reset_ET01 )
      wire#w1
      S_SR(operand := #DesApil_ET00, r1 := wire#w2)
   END_RUNG
   RUNG wire#powerrail
      Contact( #DesApil_ET08 )
      Contact( #GarrasAbiertas )
      I_Contact( #OrdenDesApilar )
      I_Contact( #OrdenMover )
      I_Contact( #Fin_OrdenMover )
      I_Contact( #MemoPosicionOK )
      { S7_Templates := "SrcType := UInt" } EQ_Contact(in1 := 0, in2 := #PosicionInicial)
      { S7_Templates := "SrcType := UInt" } EQ_Contact(in1 := 0, in2 := #PosicionFinal)
      { S7_Templates := "SrcType := UInt" } EQ_Contact(in1 := 0, in2 := #TipoAmarre)
   END_RUNG wire#w1
   RUNG wire#powerrail
      Contact( #Reset_ET01 )
      Contact( #CentradoresAbiertos )
      Contact( #GarrasAbiertas )
      Contact( #EstadoZona.Marcha_CBx )
      I_Contact( #EstadoZona.PerReset_CBx )
      I_Contact( #EstadoZona.ParoBlando_CBx )
   END_RUNG wire#w1
   RUNG wire#powerrail
      Contact( #DesApil_ET01 )
   END_RUNG wire#w2
   RUNG wire#powerrail
      Contact( #Reset_ET00 )
   END_RUNG wire#w2
   // the same network as SCL:
   IF (#AuxEstados AND NOT #Reset_ET00 AND NOT #Reset_ET01) OR (#DesApil_ET08 AND #GarrasAbiertas AND NOT #OrdenDesApilar AND NOT #OrdenMover AND NOT #Fin_OrdenMover AND NOT #MemoPosicionOK AND (0 = #PosicionInicial) AND (0 = #PosicionFinal) AND (0 = #TipoAmarre)) OR (#Reset_ET01 AND #CentradoresAbiertos AND #GarrasAbiertas AND #EstadoZona.Marcha_CBx AND NOT #EstadoZona.PerReset_CBx AND NOT #EstadoZona.ParoBlando_CBx) THEN
       #DesApil_ET00 := TRUE;   // SR flip-flop
   END_IF;
   IF #DesApil_ET01 OR #Reset_ET00 THEN #DesApil_ET00 := FALSE; END_IF;
END_REGION

REGION Network 30: VARIABLES AUXILIARES - Fin de Reset
   RUNG wire#powerrail
      Contact( #Reset_ET00 )
      Contact( #EstadoZona.PerReset_CBx )
      wire#w1
      Coil( #EstadoMAQ.Fin_VI )
   END_RUNG
   RUNG wire#powerrail
      Contact( #DesApil_ET00 )
      Contact( #MAQx_DesHabilitada )
   END_RUNG wire#w1
   // the same network as SCL:
   #EstadoMAQ.Fin_VI := (#Reset_ET00 AND #EstadoZona.PerReset_CBx) OR (#DesApil_ET00 AND #MAQx_DesHabilitada);
END_REGION

REGION Network 31: VARIABLES AUXILIARES - Fin de Paro Blando
   RUNG wire#powerrail
      Contact( #DesApil_ET00 )
      wire#w1
      Contact( #EstadoZona.ParoBlando_CBx )
      Coil( #EstadoMAQ.Paro_Blando )
   END_RUNG
   RUNG wire#powerrail
      Contact( #EstadoZona.Paro_CBx )
   END_RUNG wire#w1
   // the same network as SCL:
   #EstadoMAQ.Paro_Blando := (#DesApil_ET00 OR #EstadoZona.Paro_CBx) AND #EstadoZona.ParoBlando_CBx;
END_REGION

REGION Network 32: VARIABLES AUXILIARES - OPERACION Posicion Inicial
   RUNG wire#powerrail
      Contact( #DesApil_ET01 )
      I_Contact( #EnPila_UnicaFila )
      wire#w1
      I_Contact( #Fin_OrdenMover )
      I_Contact( #Carga_PosicionInicial )
      I_Contact( #Carga_PosicionIntermedia )
      I_Contact( #Carga_PosicionFinal )
      I_Contact( #Carga_PosicionManual )
      S_SR(operand := #Carga_PosicionInicial, r1 := wire#w2)
   END_RUNG
   RUNG wire#powerrail
      Contact( #DesApil_ET02 )
   END_RUNG wire#w1
   RUNG wire#powerrail
      I_Contact( #DesApil_ET01 )
      I_Contact( #DesApil_ET02 )
   END_RUNG wire#w2
   // the same network as SCL:
   IF ((#DesApil_ET01 AND NOT #EnPila_UnicaFila) OR #DesApil_ET02) AND NOT #Fin_OrdenMover AND NOT #Carga_PosicionInicial AND NOT #Carga_PosicionIntermedia AND NOT #Carga_PosicionFinal AND NOT #Carga_PosicionManual THEN
       #Carga_PosicionInicial := TRUE;   // SR flip-flop
   END_IF;
   IF NOT #DesApil_ET01 AND NOT #DesApil_ET02 THEN #Carga_PosicionInicial := FALSE; END_IF;
END_REGION

REGION Network 33: VARIABLES AUXILIARES - OPERACION Posicion Intermedia
   RUNG wire#powerrail
      Contact( #DesApil_ET03 )
      wire#w1
      I_Contact( #Fin_OrdenMover )
      I_Contact( #Carga_PosicionInicial )
      I_Contact( #Carga_PosicionIntermedia )
      I_Contact( #Carga_PosicionFinal )
      I_Contact( #Carga_PosicionManual )
      S_SR(operand := #Carga_PosicionIntermedia, r1 := wire#w2)
   END_RUNG
   RUNG wire#powerrail
      Contact( #DesApil_ET04 )
   END_RUNG wire#w1
   RUNG wire#powerrail
      Contact( #DesApil_ET01 )
      Contact( #EnPila_UnicaFila )
   END_RUNG wire#w1
   RUNG wire#powerrail
      I_Contact( #DesApil_ET03 )
      I_Contact( #DesApil_ET04 )
      I_Contact( #DesApil_ET01 )
   END_RUNG wire#w2
   // the same network as SCL:
   IF (#DesApil_ET03 OR #DesApil_ET04 OR (#DesApil_ET01 AND #EnPila_UnicaFila)) AND NOT #Fin_OrdenMover AND NOT #Carga_PosicionInicial AND NOT #Carga_PosicionIntermedia AND NOT #Carga_PosicionFinal AND NOT #Carga_PosicionManual THEN
       #Carga_PosicionIntermedia := TRUE;   // SR flip-flop
   END_IF;
   IF NOT #DesApil_ET03 AND NOT #DesApil_ET04 AND NOT #DesApil_ET01 THEN
       #Carga_PosicionIntermedia := FALSE;
   END_IF;
END_REGION

REGION Network 34: VARIABLES AUXILIARES - OPERACION Posicion Final
   RUNG wire#powerrail
      Contact( #DesApil_ET06 )
      wire#w1
      I_Contact( #Fin_OrdenMover )
      I_Contact( #Carga_PosicionInicial )
      I_Contact( #Carga_PosicionIntermedia )
      I_Contact( #Carga_PosicionFinal )
      I_Contact( #Carga_PosicionManual )
      S_SR(operand := #Carga_PosicionFinal, r1 := wire#w2)
   END_RUNG
   RUNG wire#powerrail
      Contact( #DesApil_ET07 )
   END_RUNG wire#w1
   RUNG wire#powerrail
      I_Contact( #DesApil_ET06 )
      I_Contact( #DesApil_ET07 )
   END_RUNG wire#w2
   // the same network as SCL:
   IF (#DesApil_ET06 OR #DesApil_ET07) AND NOT #Fin_OrdenMover AND NOT #Carga_PosicionInicial AND NOT #Carga_PosicionIntermedia AND NOT #Carga_PosicionFinal AND NOT #Carga_PosicionManual THEN
       #Carga_PosicionFinal := TRUE;   // SR flip-flop
   END_IF;
   IF NOT #DesApil_ET06 AND NOT #DesApil_ET07 THEN #Carga_PosicionFinal := FALSE; END_IF;
END_REGION

REGION Network 35: VARIABLES AUXILIARES - OPERACION Posicion Manual
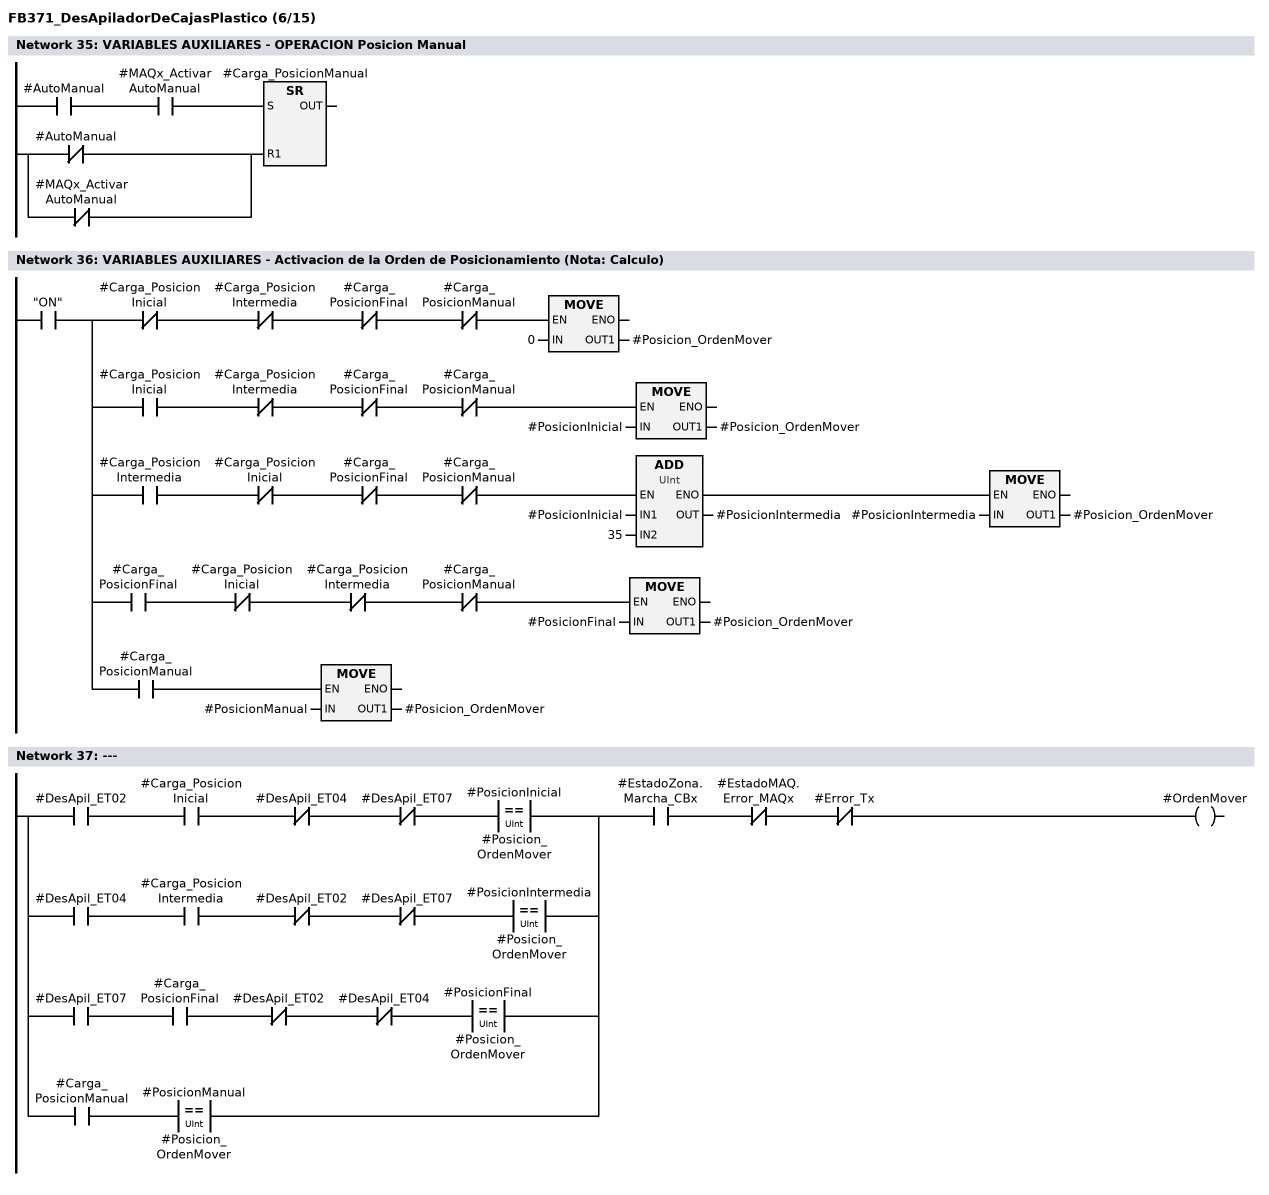
   RUNG wire#powerrail
      Contact( #AutoManual )
      Contact( #MAQx_ActivarAutoManual )
      S_SR(operand := #Carga_PosicionManual, r1 := wire#w1)
   END_RUNG
   RUNG wire#powerrail
      I_Contact( #AutoManual )
   END_RUNG wire#w1
   RUNG wire#powerrail
      I_Contact( #MAQx_ActivarAutoManual )
   END_RUNG wire#w1
   // the same network as SCL:
   IF #AutoManual AND #MAQx_ActivarAutoManual THEN
       #Carga_PosicionManual := TRUE;   // SR flip-flop
   END_IF;
   IF NOT #AutoManual OR NOT #MAQx_ActivarAutoManual THEN #Carga_PosicionManual := FALSE; END_IF;
END_REGION

REGION Network 36: VARIABLES AUXILIARES - Activacion de la Orden de Posicionamiento (Nota: Calculo)
   RUNG wire#powerrail
      Contact( "ON" )
      wire#w1
      I_Contact( #Carga_PosicionInicial )
      I_Contact( #Carga_PosicionIntermedia )
      I_Contact( #Carga_PosicionFinal )
      I_Contact( #Carga_PosicionManual )
      { S7_GenerateENO := "TRUE" } Move(in := 0, out1 => #Posicion_OrdenMover)
   END_RUNG
   RUNG wire#w1
      Contact( #Carga_PosicionInicial )
      I_Contact( #Carga_PosicionIntermedia )
      I_Contact( #Carga_PosicionFinal )
      I_Contact( #Carga_PosicionManual )
      { S7_GenerateENO := "TRUE" } Move(in := #PosicionInicial, out1 => #Posicion_OrdenMover)
   END_RUNG
   RUNG wire#w1
      Contact( #Carga_PosicionIntermedia )
      I_Contact( #Carga_PosicionInicial )
      I_Contact( #Carga_PosicionFinal )
      I_Contact( #Carga_PosicionManual )
      { S7_Templates := "SrcType := UInt"; S7_GenerateENO := "TRUE" } Add(in1 := #PosicionInicial, in2 := 35, out => #PosicionIntermedia)
      { S7_GenerateENO := "TRUE" } Move(in := #PosicionIntermedia, out1 => #Posicion_OrdenMover)
   END_RUNG
   RUNG wire#w1
      Contact( #Carga_PosicionFinal )
      I_Contact( #Carga_PosicionInicial )
      I_Contact( #Carga_PosicionIntermedia )
      I_Contact( #Carga_PosicionManual )
      { S7_GenerateENO := "TRUE" } Move(in := #PosicionFinal, out1 => #Posicion_OrdenMover)
   END_RUNG
   RUNG wire#w1
      Contact( #Carga_PosicionManual )
      { S7_GenerateENO := "TRUE" } Move(in := #PosicionManual, out1 => #Posicion_OrdenMover)
   END_RUNG
   // the same network as SCL:
   // ENO of a box is taken as its EN; it also drops when the box reports an error
   IF "ON" AND NOT #Carga_PosicionInicial AND NOT #Carga_PosicionIntermedia AND NOT #Carga_PosicionFinal AND NOT #Carga_PosicionManual THEN
       #Posicion_OrdenMover := 0;
   END_IF;
   IF "ON" AND #Carga_PosicionInicial AND NOT #Carga_PosicionIntermedia AND NOT #Carga_PosicionFinal AND NOT #Carga_PosicionManual THEN
       #Posicion_OrdenMover := #PosicionInicial;
   END_IF;
   IF "ON" AND #Carga_PosicionIntermedia AND NOT #Carga_PosicionInicial AND NOT #Carga_PosicionFinal AND NOT #Carga_PosicionManual THEN
       #PosicionIntermedia := #PosicionInicial + 35;
       #Posicion_OrdenMover := #PosicionIntermedia;
   END_IF;
   IF "ON" AND #Carga_PosicionFinal AND NOT #Carga_PosicionInicial AND NOT #Carga_PosicionIntermedia AND NOT #Carga_PosicionManual THEN
       #Posicion_OrdenMover := #PosicionFinal;
   END_IF;
   IF "ON" AND #Carga_PosicionManual THEN #Posicion_OrdenMover := #PosicionManual; END_IF;
END_REGION

REGION Network 37: ---
   RUNG wire#powerrail
      Contact( #DesApil_ET02 )
      Contact( #Carga_PosicionInicial )
      I_Contact( #DesApil_ET04 )
      I_Contact( #DesApil_ET07 )
      { S7_Templates := "SrcType := UInt" } EQ_Contact(in1 := #PosicionInicial, in2 := #Posicion_OrdenMover)
      wire#w1
      Contact( #EstadoZona.Marcha_CBx )
      I_Contact( #EstadoMAQ.Error_MAQx )
      I_Contact( #Error_Tx )
      Coil( #OrdenMover )
   END_RUNG
   RUNG wire#powerrail
      Contact( #DesApil_ET04 )
      Contact( #Carga_PosicionIntermedia )
      I_Contact( #DesApil_ET02 )
      I_Contact( #DesApil_ET07 )
      { S7_Templates := "SrcType := UInt" } EQ_Contact(in1 := #PosicionIntermedia, in2 := #Posicion_OrdenMover)
   END_RUNG wire#w1
   RUNG wire#powerrail
      Contact( #DesApil_ET07 )
      Contact( #Carga_PosicionFinal )
      I_Contact( #DesApil_ET02 )
      I_Contact( #DesApil_ET04 )
      { S7_Templates := "SrcType := UInt" } EQ_Contact(in1 := #PosicionFinal, in2 := #Posicion_OrdenMover)
   END_RUNG wire#w1
   RUNG wire#powerrail
      Contact( #Carga_PosicionManual )
      { S7_Templates := "SrcType := UInt" } EQ_Contact(in1 := #PosicionManual, in2 := #Posicion_OrdenMover)
   END_RUNG wire#w1
   // the same network as SCL:
   #OrdenMover := ((#DesApil_ET02 AND #Carga_PosicionInicial AND NOT #DesApil_ET04 AND NOT #DesApil_ET07 AND (#PosicionInicial = #Posicion_OrdenMover)) OR (#DesApil_ET04 AND #Carga_PosicionIntermedia AND NOT #DesApil_ET02 AND NOT #DesApil_ET07 AND (#PosicionIntermedia = #Posicion_OrdenMover)) OR (#DesApil_ET07 AND #Carga_PosicionFinal AND NOT #DesApil_ET02 AND NOT #DesApil_ET04 AND (#PosicionFinal = #Posicion_OrdenMover)) OR (#Carga_PosicionManual AND (#PosicionManual = #Posicion_OrdenMover))) AND #EstadoZona.Marcha_CBx AND NOT #EstadoMAQ.Error_MAQx AND NOT #Error_Tx;
END_REGION

REGION Network 38: INTERLOCK - Mesa del DesApilador de Cajas de Plastico
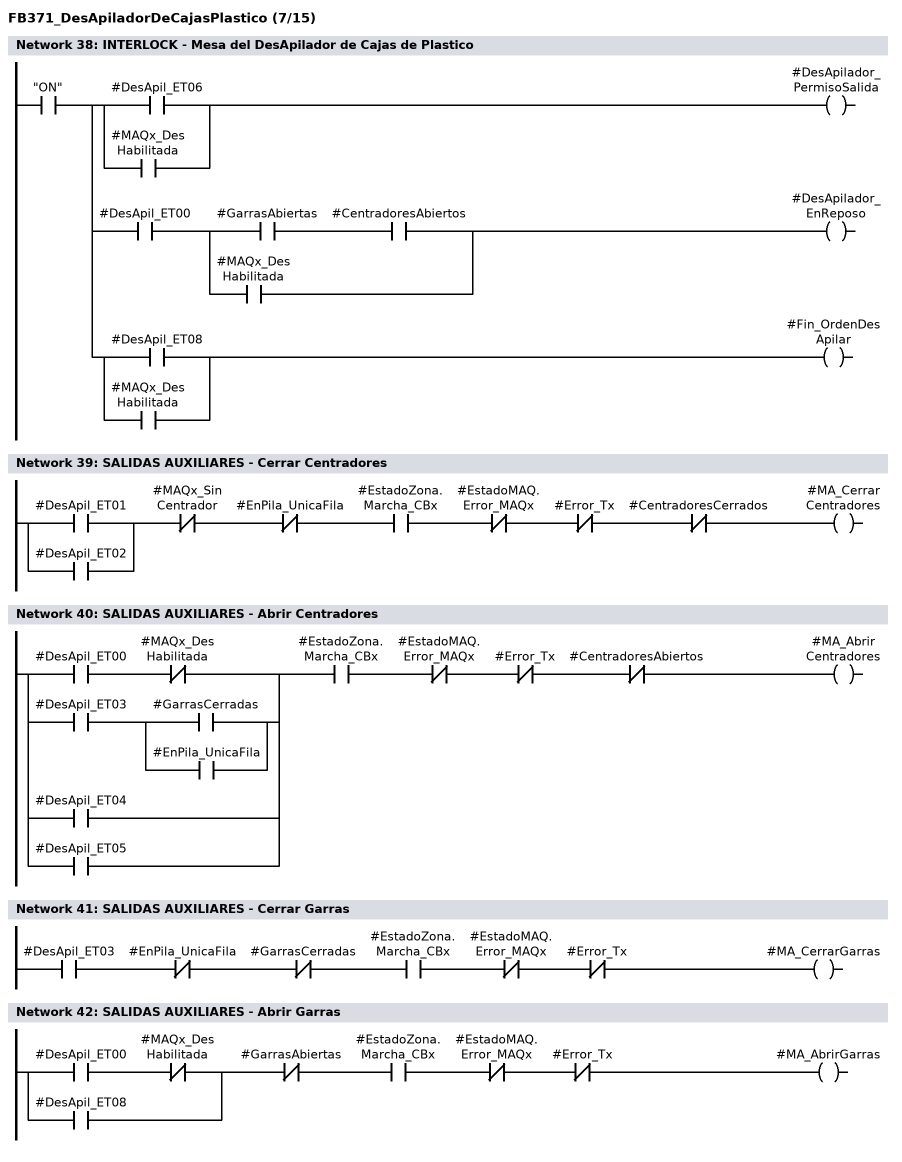
   RUNG wire#powerrail
      Contact( "ON" )
      wire#w1
      Contact( #DesApil_ET06 )
      wire#w2
      Coil( #DesApilador_PermisoSalida )
   END_RUNG
   RUNG wire#w1
      Contact( #MAQx_DesHabilitada )
   END_RUNG wire#w2
   RUNG wire#w1
      Contact( #DesApil_ET00 )
      wire#w3
      Contact( #GarrasAbiertas )
      Contact( #CentradoresAbiertos )
      wire#w4
      Coil( #DesApilador_EnReposo )
   END_RUNG
   RUNG wire#w3
      Contact( #MAQx_DesHabilitada )
   END_RUNG wire#w4
   RUNG wire#w1
      Contact( #DesApil_ET08 )
      wire#w5
      Coil( #Fin_OrdenDesApilar )
   END_RUNG
   RUNG wire#w1
      Contact( #MAQx_DesHabilitada )
   END_RUNG wire#w5
   // the same network as SCL:
   #DesApilador_PermisoSalida := "ON" AND (#DesApil_ET06 OR #MAQx_DesHabilitada);
   #DesApilador_EnReposo := "ON" AND #DesApil_ET00 AND ((#GarrasAbiertas AND #CentradoresAbiertos) OR #MAQx_DesHabilitada);
   #Fin_OrdenDesApilar := "ON" AND (#DesApil_ET08 OR #MAQx_DesHabilitada);
END_REGION

REGION Network 39: SALIDAS AUXILIARES - Cerrar Centradores
   RUNG wire#powerrail
      Contact( #DesApil_ET01 )
      wire#w1
      I_Contact( #MAQx_SinCentrador )
      I_Contact( #EnPila_UnicaFila )
      Contact( #EstadoZona.Marcha_CBx )
      I_Contact( #EstadoMAQ.Error_MAQx )
      I_Contact( #Error_Tx )
      I_Contact( #CentradoresCerrados )
      Coil( #MA_CerrarCentradores )
   END_RUNG
   RUNG wire#powerrail
      Contact( #DesApil_ET02 )
   END_RUNG wire#w1
   // the same network as SCL:
   #MA_CerrarCentradores := (#DesApil_ET01 OR #DesApil_ET02) AND NOT #MAQx_SinCentrador AND NOT #EnPila_UnicaFila AND #EstadoZona.Marcha_CBx AND NOT #EstadoMAQ.Error_MAQx AND NOT #Error_Tx AND NOT #CentradoresCerrados;
END_REGION

REGION Network 40: SALIDAS AUXILIARES - Abrir Centradores
   RUNG wire#powerrail
      Contact( #DesApil_ET00 )
      I_Contact( #MAQx_DesHabilitada )
      wire#w1
      Contact( #EstadoZona.Marcha_CBx )
      I_Contact( #EstadoMAQ.Error_MAQx )
      I_Contact( #Error_Tx )
      I_Contact( #CentradoresAbiertos )
      Coil( #MA_AbrirCentradores )
   END_RUNG
   RUNG wire#powerrail
      Contact( #DesApil_ET03 )
      wire#w2
      Contact( #GarrasCerradas )
   END_RUNG wire#w1
   RUNG wire#w2
      Contact( #EnPila_UnicaFila )
   END_RUNG wire#w1
   RUNG wire#powerrail
      Contact( #DesApil_ET04 )
   END_RUNG wire#w1
   RUNG wire#powerrail
      Contact( #DesApil_ET05 )
   END_RUNG wire#w1
   // the same network as SCL:
   #MA_AbrirCentradores := ((#DesApil_ET00 AND NOT #MAQx_DesHabilitada) OR (#DesApil_ET03 AND (#GarrasCerradas OR #EnPila_UnicaFila)) OR #DesApil_ET04 OR #DesApil_ET05) AND #EstadoZona.Marcha_CBx AND NOT #EstadoMAQ.Error_MAQx AND NOT #Error_Tx AND NOT #CentradoresAbiertos;
END_REGION

REGION Network 41: SALIDAS AUXILIARES - Cerrar Garras
   RUNG wire#powerrail
      Contact( #DesApil_ET03 )
      I_Contact( #EnPila_UnicaFila )
      I_Contact( #GarrasCerradas )
      Contact( #EstadoZona.Marcha_CBx )
      I_Contact( #EstadoMAQ.Error_MAQx )
      I_Contact( #Error_Tx )
      Coil( #MA_CerrarGarras )
   END_RUNG
   // the same network as SCL:
   #MA_CerrarGarras := #DesApil_ET03 AND NOT #EnPila_UnicaFila AND NOT #GarrasCerradas AND #EstadoZona.Marcha_CBx AND NOT #EstadoMAQ.Error_MAQx AND NOT #Error_Tx;
END_REGION

REGION Network 42: SALIDAS AUXILIARES - Abrir Garras
   RUNG wire#powerrail
      Contact( #DesApil_ET00 )
      I_Contact( #MAQx_DesHabilitada )
      wire#w1
      I_Contact( #GarrasAbiertas )
      Contact( #EstadoZona.Marcha_CBx )
      I_Contact( #EstadoMAQ.Error_MAQx )
      I_Contact( #Error_Tx )
      Coil( #MA_AbrirGarras )
   END_RUNG
   RUNG wire#powerrail
      Contact( #DesApil_ET08 )
   END_RUNG wire#w1
   // the same network as SCL:
   #MA_AbrirGarras := ((#DesApil_ET00 AND NOT #MAQx_DesHabilitada) OR #DesApil_ET08) AND NOT #GarrasAbiertas AND #EstadoZona.Marcha_CBx AND NOT #EstadoMAQ.Error_MAQx AND NOT #Error_Tx;
END_REGION

REGION Network 43: SALIDAS AUXILIARES - Cerrar Guias
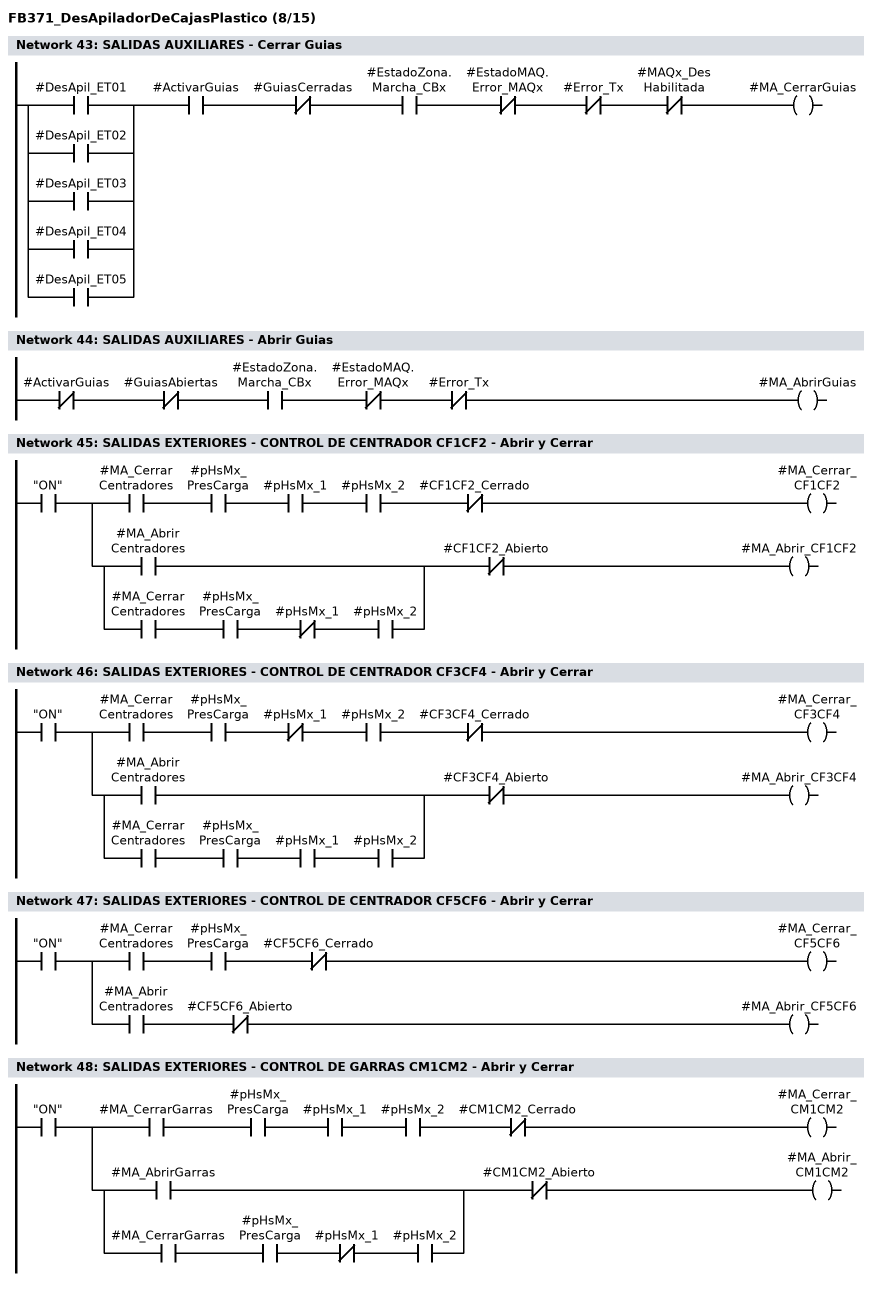
   RUNG wire#powerrail
      Contact( #DesApil_ET01 )
      wire#w1
      Contact( #ActivarGuias )
      I_Contact( #GuiasCerradas )
      Contact( #EstadoZona.Marcha_CBx )
      I_Contact( #EstadoMAQ.Error_MAQx )
      I_Contact( #Error_Tx )
      I_Contact( #MAQx_DesHabilitada )
      Coil( #MA_CerrarGuias )
   END_RUNG
   RUNG wire#powerrail
      Contact( #DesApil_ET02 )
   END_RUNG wire#w1
   RUNG wire#powerrail
      Contact( #DesApil_ET03 )
   END_RUNG wire#w1
   RUNG wire#powerrail
      Contact( #DesApil_ET04 )
   END_RUNG wire#w1
   RUNG wire#powerrail
      Contact( #DesApil_ET05 )
   END_RUNG wire#w1
   // the same network as SCL:
   #MA_CerrarGuias := (#DesApil_ET01 OR #DesApil_ET02 OR #DesApil_ET03 OR #DesApil_ET04 OR #DesApil_ET05) AND #ActivarGuias AND NOT #GuiasCerradas AND #EstadoZona.Marcha_CBx AND NOT #EstadoMAQ.Error_MAQx AND NOT #Error_Tx AND NOT #MAQx_DesHabilitada;
END_REGION

REGION Network 44: SALIDAS AUXILIARES - Abrir Guias
   RUNG wire#powerrail
      I_Contact( #ActivarGuias )
      I_Contact( #GuiasAbiertas )
      Contact( #EstadoZona.Marcha_CBx )
      I_Contact( #EstadoMAQ.Error_MAQx )
      I_Contact( #Error_Tx )
      Coil( #MA_AbrirGuias )
   END_RUNG
   // the same network as SCL:
   #MA_AbrirGuias := NOT #ActivarGuias AND NOT #GuiasAbiertas AND #EstadoZona.Marcha_CBx AND NOT #EstadoMAQ.Error_MAQx AND NOT #Error_Tx;
END_REGION

REGION Network 45: SALIDAS EXTERIORES - CONTROL DE CENTRADOR CF1CF2 - Abrir y Cerrar
   RUNG wire#powerrail
      Contact( "ON" )
      wire#w1
      Contact( #MA_CerrarCentradores )
      Contact( #pHsMx_PresCarga )
      Contact( #pHsMx_1 )
      Contact( #pHsMx_2 )
      I_Contact( #CF1CF2_Cerrado )
      Coil( #MA_Cerrar_CF1CF2 )
   END_RUNG
   RUNG wire#w1
      Contact( #MA_AbrirCentradores )
      wire#w2
      I_Contact( #CF1CF2_Abierto )
      Coil( #MA_Abrir_CF1CF2 )
   END_RUNG
   RUNG wire#w1
      Contact( #MA_CerrarCentradores )
      Contact( #pHsMx_PresCarga )
      I_Contact( #pHsMx_1 )
      Contact( #pHsMx_2 )
   END_RUNG wire#w2
   // the same network as SCL:
   #MA_Cerrar_CF1CF2 := "ON" AND #MA_CerrarCentradores AND #pHsMx_PresCarga AND #pHsMx_1 AND #pHsMx_2 AND NOT #CF1CF2_Cerrado;
   #MA_Abrir_CF1CF2 := "ON" AND (#MA_AbrirCentradores OR (#MA_CerrarCentradores AND #pHsMx_PresCarga AND NOT #pHsMx_1 AND #pHsMx_2)) AND NOT #CF1CF2_Abierto;
END_REGION

REGION Network 46: SALIDAS EXTERIORES - CONTROL DE CENTRADOR CF3CF4 - Abrir y Cerrar
   RUNG wire#powerrail
      Contact( "ON" )
      wire#w1
      Contact( #MA_CerrarCentradores )
      Contact( #pHsMx_PresCarga )
      I_Contact( #pHsMx_1 )
      Contact( #pHsMx_2 )
      I_Contact( #CF3CF4_Cerrado )
      Coil( #MA_Cerrar_CF3CF4 )
   END_RUNG
   RUNG wire#w1
      Contact( #MA_AbrirCentradores )
      wire#w2
      I_Contact( #CF3CF4_Abierto )
      Coil( #MA_Abrir_CF3CF4 )
   END_RUNG
   RUNG wire#w1
      Contact( #MA_CerrarCentradores )
      Contact( #pHsMx_PresCarga )
      Contact( #pHsMx_1 )
      Contact( #pHsMx_2 )
   END_RUNG wire#w2
   // the same network as SCL:
   #MA_Cerrar_CF3CF4 := "ON" AND #MA_CerrarCentradores AND #pHsMx_PresCarga AND NOT #pHsMx_1 AND #pHsMx_2 AND NOT #CF3CF4_Cerrado;
   #MA_Abrir_CF3CF4 := "ON" AND (#MA_AbrirCentradores OR (#MA_CerrarCentradores AND #pHsMx_PresCarga AND #pHsMx_1 AND #pHsMx_2)) AND NOT #CF3CF4_Abierto;
END_REGION

REGION Network 47: SALIDAS EXTERIORES - CONTROL DE CENTRADOR CF5CF6 - Abrir y Cerrar
   RUNG wire#powerrail
      Contact( "ON" )
      wire#w1
      Contact( #MA_CerrarCentradores )
      Contact( #pHsMx_PresCarga )
      I_Contact( #CF5CF6_Cerrado )
      Coil( #MA_Cerrar_CF5CF6 )
   END_RUNG
   RUNG wire#w1
      Contact( #MA_AbrirCentradores )
      I_Contact( #CF5CF6_Abierto )
      Coil( #MA_Abrir_CF5CF6 )
   END_RUNG
   // the same network as SCL:
   #MA_Cerrar_CF5CF6 := "ON" AND #MA_CerrarCentradores AND #pHsMx_PresCarga AND NOT #CF5CF6_Cerrado;
   #MA_Abrir_CF5CF6 := "ON" AND #MA_AbrirCentradores AND NOT #CF5CF6_Abierto;
END_REGION

REGION Network 48: SALIDAS EXTERIORES - CONTROL DE GARRAS CM1CM2 - Abrir y Cerrar
   RUNG wire#powerrail
      Contact( "ON" )
      wire#w1
      Contact( #MA_CerrarGarras )
      Contact( #pHsMx_PresCarga )
      Contact( #pHsMx_1 )
      Contact( #pHsMx_2 )
      I_Contact( #CM1CM2_Cerrado )
      Coil( #MA_Cerrar_CM1CM2 )
   END_RUNG
   RUNG wire#w1
      Contact( #MA_AbrirGarras )
      wire#w2
      I_Contact( #CM1CM2_Abierto )
      Coil( #MA_Abrir_CM1CM2 )
   END_RUNG
   RUNG wire#w1
      Contact( #MA_CerrarGarras )
      Contact( #pHsMx_PresCarga )
      I_Contact( #pHsMx_1 )
      Contact( #pHsMx_2 )
   END_RUNG wire#w2
   // the same network as SCL:
   #MA_Cerrar_CM1CM2 := "ON" AND #MA_CerrarGarras AND #pHsMx_PresCarga AND #pHsMx_1 AND #pHsMx_2 AND NOT #CM1CM2_Cerrado;
   #MA_Abrir_CM1CM2 := "ON" AND (#MA_AbrirGarras OR (#MA_CerrarGarras AND #pHsMx_PresCarga AND NOT #pHsMx_1 AND #pHsMx_2)) AND NOT #CM1CM2_Abierto;
END_REGION

REGION Network 49: SALIDAS EXTERIORES - CONTROL DE GARRAS CM3CM4 - Abrir y Cerrar >>> Caja EuroPool CM3CM8
   // Nota: Caja Tipo Europool >>> Utilizar para Caja Pequeña
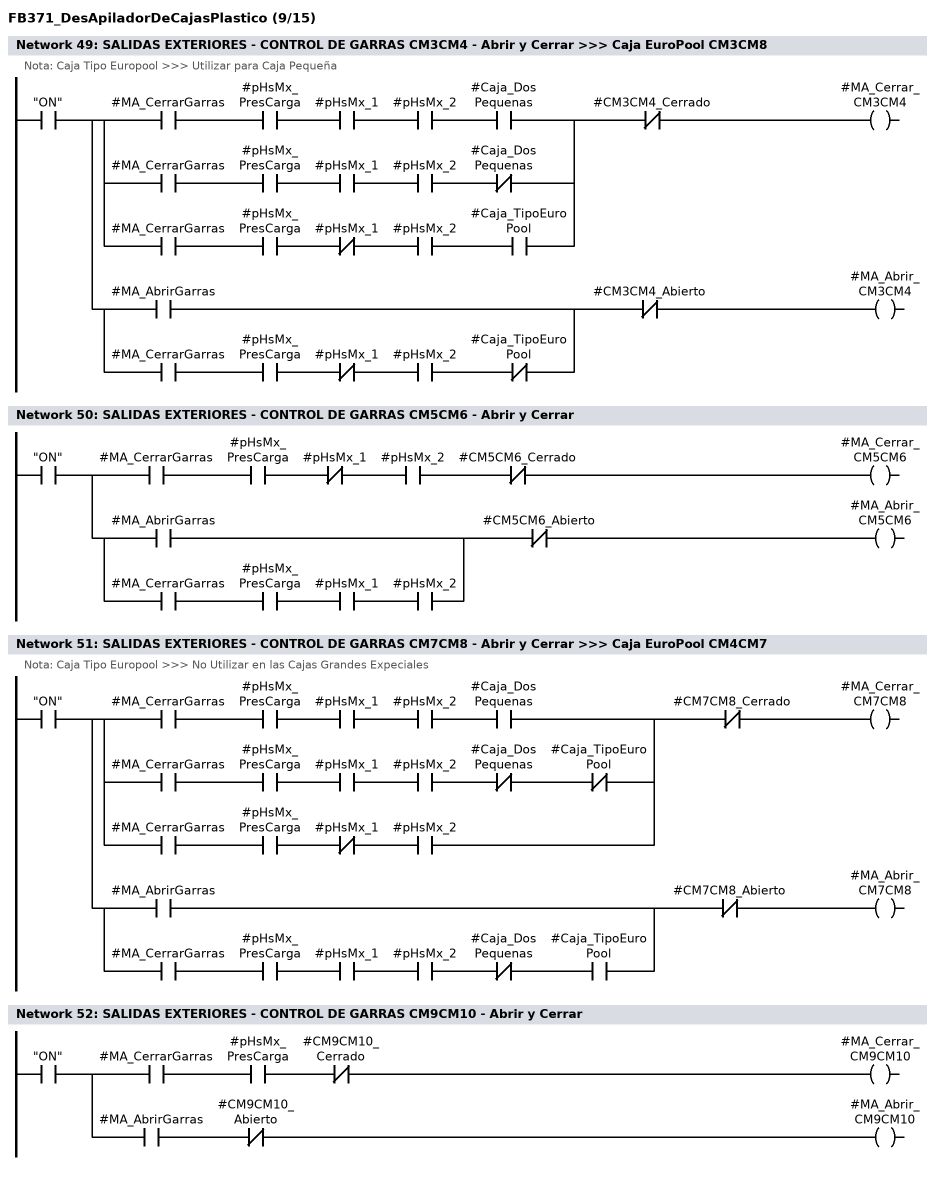
   RUNG wire#powerrail
      Contact( "ON" )
      wire#w1
      Contact( #MA_CerrarGarras )
      Contact( #pHsMx_PresCarga )
      Contact( #pHsMx_1 )
      Contact( #pHsMx_2 )
      Contact( #Caja_DosPequenas )
      wire#w2
      I_Contact( #CM3CM4_Cerrado )
      Coil( #MA_Cerrar_CM3CM4 )
   END_RUNG
   RUNG wire#w1
      Contact( #MA_CerrarGarras )
      Contact( #pHsMx_PresCarga )
      Contact( #pHsMx_1 )
      Contact( #pHsMx_2 )
      I_Contact( #Caja_DosPequenas )
   END_RUNG wire#w2
   RUNG wire#w1
      Contact( #MA_CerrarGarras )
      Contact( #pHsMx_PresCarga )
      I_Contact( #pHsMx_1 )
      Contact( #pHsMx_2 )
      Contact( #Caja_TipoEuroPool )
   END_RUNG wire#w2
   RUNG wire#w1
      Contact( #MA_AbrirGarras )
      wire#w3
      I_Contact( #CM3CM4_Abierto )
      Coil( #MA_Abrir_CM3CM4 )
   END_RUNG
   RUNG wire#w1
      Contact( #MA_CerrarGarras )
      Contact( #pHsMx_PresCarga )
      I_Contact( #pHsMx_1 )
      Contact( #pHsMx_2 )
      I_Contact( #Caja_TipoEuroPool )
   END_RUNG wire#w3
   // the same network as SCL:
   #MA_Cerrar_CM3CM4 := "ON" AND ((#MA_CerrarGarras AND #pHsMx_PresCarga AND #pHsMx_1 AND #pHsMx_2 AND #Caja_DosPequenas) OR (#MA_CerrarGarras AND #pHsMx_PresCarga AND #pHsMx_1 AND #pHsMx_2 AND NOT #Caja_DosPequenas) OR (#MA_CerrarGarras AND #pHsMx_PresCarga AND NOT #pHsMx_1 AND #pHsMx_2 AND #Caja_TipoEuroPool)) AND NOT #CM3CM4_Cerrado;
   #MA_Abrir_CM3CM4 := "ON" AND (#MA_AbrirGarras OR (#MA_CerrarGarras AND #pHsMx_PresCarga AND NOT #pHsMx_1 AND #pHsMx_2 AND NOT #Caja_TipoEuroPool)) AND NOT #CM3CM4_Abierto;
END_REGION

REGION Network 50: SALIDAS EXTERIORES - CONTROL DE GARRAS CM5CM6 - Abrir y Cerrar
   RUNG wire#powerrail
      Contact( "ON" )
      wire#w1
      Contact( #MA_CerrarGarras )
      Contact( #pHsMx_PresCarga )
      I_Contact( #pHsMx_1 )
      Contact( #pHsMx_2 )
      I_Contact( #CM5CM6_Cerrado )
      Coil( #MA_Cerrar_CM5CM6 )
   END_RUNG
   RUNG wire#w1
      Contact( #MA_AbrirGarras )
      wire#w2
      I_Contact( #CM5CM6_Abierto )
      Coil( #MA_Abrir_CM5CM6 )
   END_RUNG
   RUNG wire#w1
      Contact( #MA_CerrarGarras )
      Contact( #pHsMx_PresCarga )
      Contact( #pHsMx_1 )
      Contact( #pHsMx_2 )
   END_RUNG wire#w2
   // the same network as SCL:
   #MA_Cerrar_CM5CM6 := "ON" AND #MA_CerrarGarras AND #pHsMx_PresCarga AND NOT #pHsMx_1 AND #pHsMx_2 AND NOT #CM5CM6_Cerrado;
   #MA_Abrir_CM5CM6 := "ON" AND (#MA_AbrirGarras OR (#MA_CerrarGarras AND #pHsMx_PresCarga AND #pHsMx_1 AND #pHsMx_2)) AND NOT #CM5CM6_Abierto;
END_REGION

REGION Network 51: SALIDAS EXTERIORES - CONTROL DE GARRAS CM7CM8 - Abrir y Cerrar >>> Caja EuroPool CM4CM7
   // Nota: Caja Tipo Europool >>> No Utilizar en las Cajas Grandes Expeciales
   RUNG wire#powerrail
      Contact( "ON" )
      wire#w1
      Contact( #MA_CerrarGarras )
      Contact( #pHsMx_PresCarga )
      Contact( #pHsMx_1 )
      Contact( #pHsMx_2 )
      Contact( #Caja_DosPequenas )
      wire#w2
      I_Contact( #CM7CM8_Cerrado )
      Coil( #MA_Cerrar_CM7CM8 )
   END_RUNG
   RUNG wire#w1
      Contact( #MA_CerrarGarras )
      Contact( #pHsMx_PresCarga )
      Contact( #pHsMx_1 )
      Contact( #pHsMx_2 )
      I_Contact( #Caja_DosPequenas )
      I_Contact( #Caja_TipoEuroPool )
   END_RUNG wire#w2
   RUNG wire#w1
      Contact( #MA_CerrarGarras )
      Contact( #pHsMx_PresCarga )
      I_Contact( #pHsMx_1 )
      Contact( #pHsMx_2 )
   END_RUNG wire#w2
   RUNG wire#w1
      Contact( #MA_AbrirGarras )
      wire#w3
      I_Contact( #CM7CM8_Abierto )
      Coil( #MA_Abrir_CM7CM8 )
   END_RUNG
   RUNG wire#w1
      Contact( #MA_CerrarGarras )
      Contact( #pHsMx_PresCarga )
      Contact( #pHsMx_1 )
      Contact( #pHsMx_2 )
      I_Contact( #Caja_DosPequenas )
      Contact( #Caja_TipoEuroPool )
   END_RUNG wire#w3
   // the same network as SCL:
   #MA_Cerrar_CM7CM8 := "ON" AND ((#MA_CerrarGarras AND #pHsMx_PresCarga AND #pHsMx_1 AND #pHsMx_2 AND #Caja_DosPequenas) OR (#MA_CerrarGarras AND #pHsMx_PresCarga AND #pHsMx_1 AND #pHsMx_2 AND NOT #Caja_DosPequenas AND NOT #Caja_TipoEuroPool) OR (#MA_CerrarGarras AND #pHsMx_PresCarga AND NOT #pHsMx_1 AND #pHsMx_2)) AND NOT #CM7CM8_Cerrado;
   #MA_Abrir_CM7CM8 := "ON" AND (#MA_AbrirGarras OR (#MA_CerrarGarras AND #pHsMx_PresCarga AND #pHsMx_1 AND #pHsMx_2 AND NOT #Caja_DosPequenas AND #Caja_TipoEuroPool)) AND NOT #CM7CM8_Abierto;
END_REGION

REGION Network 52: SALIDAS EXTERIORES - CONTROL DE GARRAS CM9CM10 - Abrir y Cerrar
   RUNG wire#powerrail
      Contact( "ON" )
      wire#w1
      Contact( #MA_CerrarGarras )
      Contact( #pHsMx_PresCarga )
      I_Contact( #CM9CM10_Cerrado )
      Coil( #MA_Cerrar_CM9CM10 )
   END_RUNG
   RUNG wire#w1
      Contact( #MA_AbrirGarras )
      I_Contact( #CM9CM10_Abierto )
      Coil( #MA_Abrir_CM9CM10 )
   END_RUNG
   // the same network as SCL:
   #MA_Cerrar_CM9CM10 := "ON" AND #MA_CerrarGarras AND #pHsMx_PresCarga AND NOT #CM9CM10_Cerrado;
   #MA_Abrir_CM9CM10 := "ON" AND #MA_AbrirGarras AND NOT #CM9CM10_Abierto;
END_REGION

REGION Network 53: SALIDAS EXTERIORES - CONTROL DE GUIAS GF1GF2 - Abrir y Cerrar
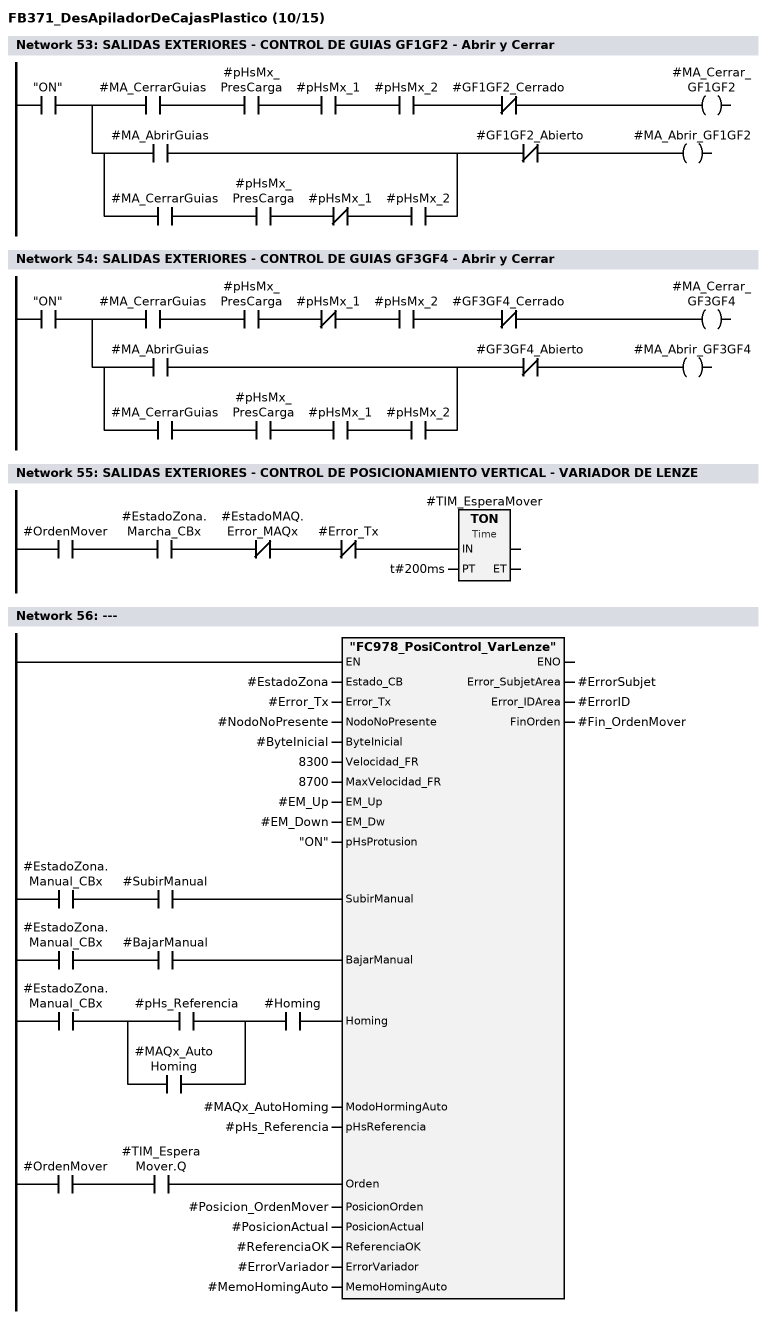
   RUNG wire#powerrail
      Contact( "ON" )
      wire#w1
      Contact( #MA_CerrarGuias )
      Contact( #pHsMx_PresCarga )
      Contact( #pHsMx_1 )
      Contact( #pHsMx_2 )
      I_Contact( #GF1GF2_Cerrado )
      Coil( #MA_Cerrar_GF1GF2 )
   END_RUNG
   RUNG wire#w1
      Contact( #MA_AbrirGuias )
      wire#w2
      I_Contact( #GF1GF2_Abierto )
      Coil( #MA_Abrir_GF1GF2 )
   END_RUNG
   RUNG wire#w1
      Contact( #MA_CerrarGuias )
      Contact( #pHsMx_PresCarga )
      I_Contact( #pHsMx_1 )
      Contact( #pHsMx_2 )
   END_RUNG wire#w2
   // the same network as SCL:
   #MA_Cerrar_GF1GF2 := "ON" AND #MA_CerrarGuias AND #pHsMx_PresCarga AND #pHsMx_1 AND #pHsMx_2 AND NOT #GF1GF2_Cerrado;
   #MA_Abrir_GF1GF2 := "ON" AND (#MA_AbrirGuias OR (#MA_CerrarGuias AND #pHsMx_PresCarga AND NOT #pHsMx_1 AND #pHsMx_2)) AND NOT #GF1GF2_Abierto;
END_REGION

REGION Network 54: SALIDAS EXTERIORES - CONTROL DE GUIAS GF3GF4 - Abrir y Cerrar
   RUNG wire#powerrail
      Contact( "ON" )
      wire#w1
      Contact( #MA_CerrarGuias )
      Contact( #pHsMx_PresCarga )
      I_Contact( #pHsMx_1 )
      Contact( #pHsMx_2 )
      I_Contact( #GF3GF4_Cerrado )
      Coil( #MA_Cerrar_GF3GF4 )
   END_RUNG
   RUNG wire#w1
      Contact( #MA_AbrirGuias )
      wire#w2
      I_Contact( #GF3GF4_Abierto )
      Coil( #MA_Abrir_GF3GF4 )
   END_RUNG
   RUNG wire#w1
      Contact( #MA_CerrarGuias )
      Contact( #pHsMx_PresCarga )
      Contact( #pHsMx_1 )
      Contact( #pHsMx_2 )
   END_RUNG wire#w2
   // the same network as SCL:
   #MA_Cerrar_GF3GF4 := "ON" AND #MA_CerrarGuias AND #pHsMx_PresCarga AND NOT #pHsMx_1 AND #pHsMx_2 AND NOT #GF3GF4_Cerrado;
   #MA_Abrir_GF3GF4 := "ON" AND (#MA_AbrirGuias OR (#MA_CerrarGuias AND #pHsMx_PresCarga AND #pHsMx_1 AND #pHsMx_2)) AND NOT #GF3GF4_Abierto;
END_REGION

REGION Network 55: SALIDAS EXTERIORES - CONTROL DE POSICIONAMIENTO VERTICAL - VARIADOR DE LENZE
   RUNG wire#powerrail
      Contact( #OrdenMover )
      Contact( #EstadoZona.Marcha_CBx )
      I_Contact( #EstadoMAQ.Error_MAQx )
      I_Contact( #Error_Tx )
      { S7_Templates := "time_type := Time" } #TIM_EsperaMover.TON(pt := t#200ms, et =>)
   END_RUNG
   // the same network as SCL:
   #TIM_EsperaMover(IN := #OrdenMover AND #EstadoZona.Marcha_CBx AND NOT #EstadoMAQ.Error_MAQx AND NOT #Error_Tx,   // TON
                    PT := t#200ms);
END_REGION

REGION Network 56: ---
   RUNG wire#powerrail
      "FC978_PosiControl_VarLenze"(SubirManual := wire#w1, BajarManual := wire#w2, Homing := wire#w5, Orden := wire#w6, Estado_CB := #EstadoZona, Error_Tx := #Error_Tx, NodoNoPresente := #NodoNoPresente, ByteInicial := #ByteInicial, Velocidad_FR := 8300, MaxVelocidad_FR := 8700, EM_Up := #EM_Up, EM_Dw := #EM_Down, pHsProtusion := "ON", ModoHormingAuto := #MAQx_AutoHoming, pHsReferencia := #pHs_Referencia, PosicionOrden := #Posicion_OrdenMover, PosicionActual := #PosicionActual, ReferenciaOK := #ReferenciaOK, ErrorVariador := #ErrorVariador, MemoHomingAuto := #MemoHomingAuto, Error_SubjetArea => #ErrorSubjet, Error_IDArea => #ErrorID, FinOrden => #Fin_OrdenMover)
   END_RUNG
   RUNG wire#powerrail
      Contact( #EstadoZona.Manual_CBx )
      Contact( #SubirManual )
   END_RUNG wire#w1
   RUNG wire#powerrail
      Contact( #EstadoZona.Manual_CBx )
      Contact( #BajarManual )
   END_RUNG wire#w2
   RUNG wire#powerrail
      Contact( #EstadoZona.Manual_CBx )
      wire#w3
      Contact( #pHs_Referencia )
      wire#w4
      Contact( #Homing )
   END_RUNG wire#w5
   RUNG wire#w3
      Contact( #MAQx_AutoHoming )
   END_RUNG wire#w4
   RUNG wire#powerrail
      Contact( #OrdenMover )
      Contact( #TIM_EsperaMover.Q )
   END_RUNG wire#w6
   // the same network as SCL:
   "FC978_PosiControl_VarLenze"(Estado_CB := #EstadoZona,
                           Error_Tx := #Error_Tx,
                           NodoNoPresente := #NodoNoPresente,
                           ByteInicial := #ByteInicial,
                           Velocidad_FR := 8300,
                           MaxVelocidad_FR := 8700,
                           EM_Up := #EM_Up,
                           EM_Dw := #EM_Down,
                           pHsProtusion := "ON",
                           SubirManual := #EstadoZona.Manual_CBx AND #SubirManual,
                           BajarManual := #EstadoZona.Manual_CBx AND #BajarManual,
                           Homing := #EstadoZona.Manual_CBx AND (#pHs_Referencia OR #MAQx_AutoHoming) AND #Homing,
                           ModoHormingAuto := #MAQx_AutoHoming,
                           pHsReferencia := #pHs_Referencia,
                           Orden := #OrdenMover AND #TIM_EsperaMover.Q,
                           PosicionOrden := #Posicion_OrdenMover,
                           PosicionActual := #PosicionActual,
                           ReferenciaOK := #ReferenciaOK,
                           ErrorVariador := #ErrorVariador,
                           MemoHomingAuto := #MemoHomingAuto,
                           Error_SubjetArea => #ErrorSubjet,
                           Error_IDArea => #ErrorID,
                           FinOrden => #Fin_OrdenMover);
END_REGION

REGION Network 57: TMP - Espera En Tension
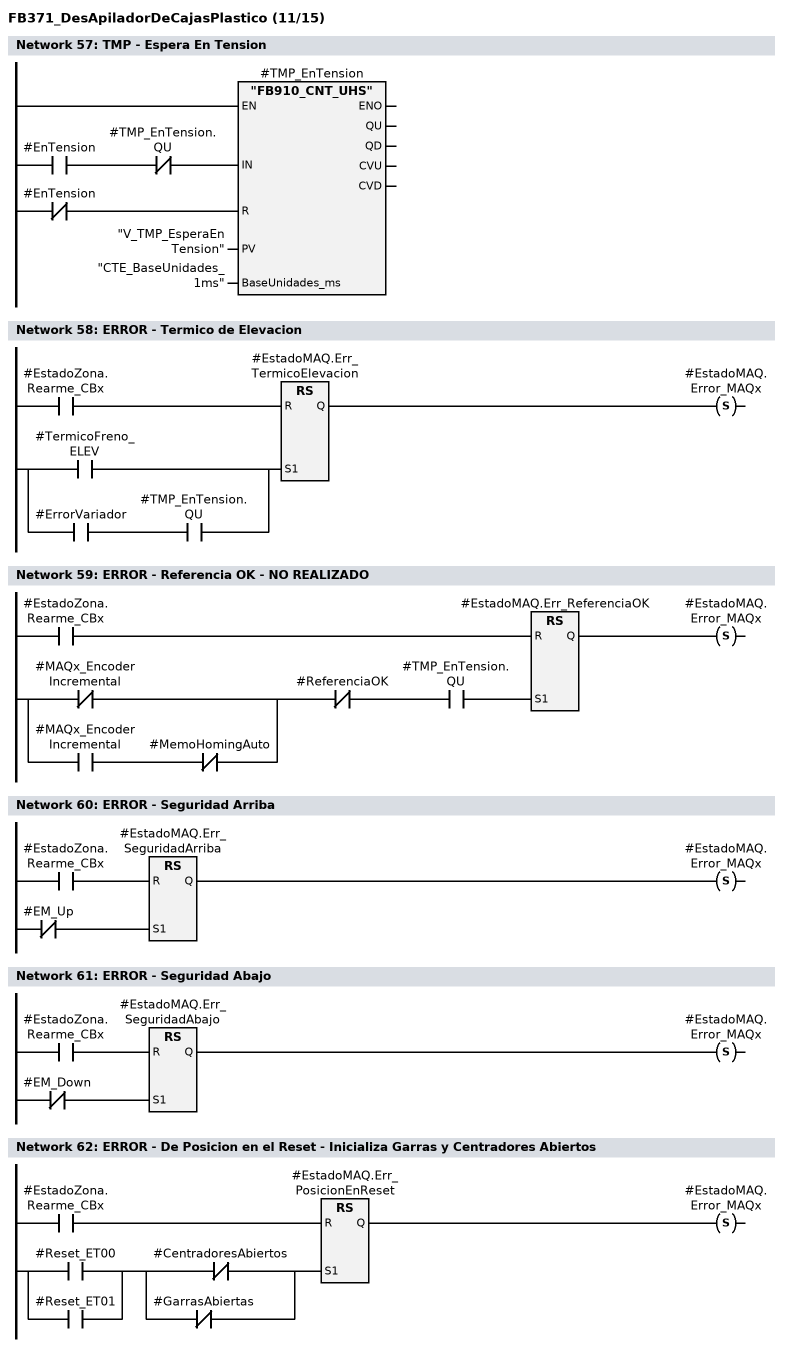
   RUNG wire#powerrail
      #TMP_EnTension(IN := wire#w1, R := wire#w2, PV := "V_TMP_EsperaEnTension", BaseUnidades_ms := "CTE_BaseUnidades_1ms", QU =>, QD =>, CVU =>, CVD =>)
   END_RUNG
   RUNG wire#powerrail
      Contact( #EnTension )
      I_Contact( #TMP_EnTension.QU )
   END_RUNG wire#w1
   RUNG wire#powerrail
      I_Contact( #EnTension )
   END_RUNG wire#w2
   // the same network as SCL:
   #TMP_EnTension(IN := #EnTension AND NOT #TMP_EnTension.QU,   // "FB910_CNT_UHS"
                  R := NOT #EnTension,
                  PV := "V_TMP_EsperaEnTension",
                  BaseUnidades_ms := "CTE_BaseUnidades_1ms");
END_REGION

REGION Network 58: ERROR - Termico de Elevacion
   RUNG wire#powerrail
      Contact( #EstadoZona.Rearme_CBx )
      S_RS(operand := #EstadoMAQ.Err_TermicoElevacion, s1 := wire#w1)
      S_Coil( #EstadoMAQ.Error_MAQx )
   END_RUNG
   RUNG wire#powerrail
      Contact( #TermicoFreno_ELEV )
   END_RUNG wire#w1
   RUNG wire#powerrail
      Contact( #ErrorVariador )
      Contact( #TMP_EnTension.QU )
   END_RUNG wire#w1
   // the same network as SCL:
   IF #EstadoZona.Rearme_CBx THEN
       #EstadoMAQ.Err_TermicoElevacion := FALSE;   // RS flip-flop
   END_IF;
   IF #TermicoFreno_ELEV OR (#ErrorVariador AND #TMP_EnTension.QU) THEN
       #EstadoMAQ.Err_TermicoElevacion := TRUE;
   END_IF;
   IF #EstadoMAQ.Err_TermicoElevacion THEN #EstadoMAQ.Error_MAQx := TRUE; END_IF;
END_REGION

REGION Network 59: ERROR - Referencia OK - NO REALIZADO
   RUNG wire#powerrail
      Contact( #EstadoZona.Rearme_CBx )
      S_RS(operand := #EstadoMAQ.Err_ReferenciaOK, s1 := wire#w2)
      S_Coil( #EstadoMAQ.Error_MAQx )
   END_RUNG
   RUNG wire#powerrail
      I_Contact( #MAQx_EncoderIncremental )
      wire#w1
      I_Contact( #ReferenciaOK )
      Contact( #TMP_EnTension.QU )
   END_RUNG wire#w2
   RUNG wire#powerrail
      Contact( #MAQx_EncoderIncremental )
      I_Contact( #MemoHomingAuto )
   END_RUNG wire#w1
   // the same network as SCL:
   IF #EstadoZona.Rearme_CBx THEN
       #EstadoMAQ.Err_ReferenciaOK := FALSE;   // RS flip-flop
   END_IF;
   IF (NOT #MAQx_EncoderIncremental OR (#MAQx_EncoderIncremental AND NOT #MemoHomingAuto)) AND NOT #ReferenciaOK AND #TMP_EnTension.QU THEN
       #EstadoMAQ.Err_ReferenciaOK := TRUE;
   END_IF;
   IF #EstadoMAQ.Err_ReferenciaOK THEN #EstadoMAQ.Error_MAQx := TRUE; END_IF;
END_REGION

REGION Network 60: ERROR - Seguridad Arriba
   RUNG wire#powerrail
      Contact( #EstadoZona.Rearme_CBx )
      S_RS(operand := #EstadoMAQ.Err_SeguridadArriba, s1 := wire#w1)
      S_Coil( #EstadoMAQ.Error_MAQx )
   END_RUNG
   RUNG wire#powerrail
      I_Contact( #EM_Up )
   END_RUNG wire#w1
   // the same network as SCL:
   IF #EstadoZona.Rearme_CBx THEN
       #EstadoMAQ.Err_SeguridadArriba := FALSE;   // RS flip-flop
   END_IF;
   IF NOT #EM_Up THEN #EstadoMAQ.Err_SeguridadArriba := TRUE; END_IF;
   IF #EstadoMAQ.Err_SeguridadArriba THEN #EstadoMAQ.Error_MAQx := TRUE; END_IF;
END_REGION

REGION Network 61: ERROR - Seguridad Abajo
   RUNG wire#powerrail
      Contact( #EstadoZona.Rearme_CBx )
      S_RS(operand := #EstadoMAQ.Err_SeguridadAbajo, s1 := wire#w1)
      S_Coil( #EstadoMAQ.Error_MAQx )
   END_RUNG
   RUNG wire#powerrail
      I_Contact( #EM_Down )
   END_RUNG wire#w1
   // the same network as SCL:
   IF #EstadoZona.Rearme_CBx THEN
       #EstadoMAQ.Err_SeguridadAbajo := FALSE;   // RS flip-flop
   END_IF;
   IF NOT #EM_Down THEN #EstadoMAQ.Err_SeguridadAbajo := TRUE; END_IF;
   IF #EstadoMAQ.Err_SeguridadAbajo THEN #EstadoMAQ.Error_MAQx := TRUE; END_IF;
END_REGION

REGION Network 62: ERROR - De Posicion en el Reset - Inicializa Garras y Centradores Abiertos
   RUNG wire#powerrail
      Contact( #EstadoZona.Rearme_CBx )
      S_RS(operand := #EstadoMAQ.Err_PosicionEnReset, s1 := wire#w2)
      S_Coil( #EstadoMAQ.Error_MAQx )
   END_RUNG
   RUNG wire#powerrail
      Contact( #Reset_ET00 )
      wire#w1
      I_Contact( #CentradoresAbiertos )
   END_RUNG wire#w2
   RUNG wire#powerrail
      Contact( #Reset_ET01 )
   END_RUNG wire#w1
   RUNG wire#w1
      I_Contact( #GarrasAbiertas )
   END_RUNG wire#w2
   // the same network as SCL:
   IF #EstadoZona.Rearme_CBx THEN
       #EstadoMAQ.Err_PosicionEnReset := FALSE;   // RS flip-flop
   END_IF;
   IF (#Reset_ET00 OR #Reset_ET01) AND (NOT #CentradoresAbiertos OR NOT #GarrasAbiertas) THEN
       #EstadoMAQ.Err_PosicionEnReset := TRUE;
   END_IF;
   IF #EstadoMAQ.Err_PosicionEnReset THEN #EstadoMAQ.Error_MAQx := TRUE; END_IF;
END_REGION

REGION Network 63: TMP - ERROR - TimeOut de Elevacion
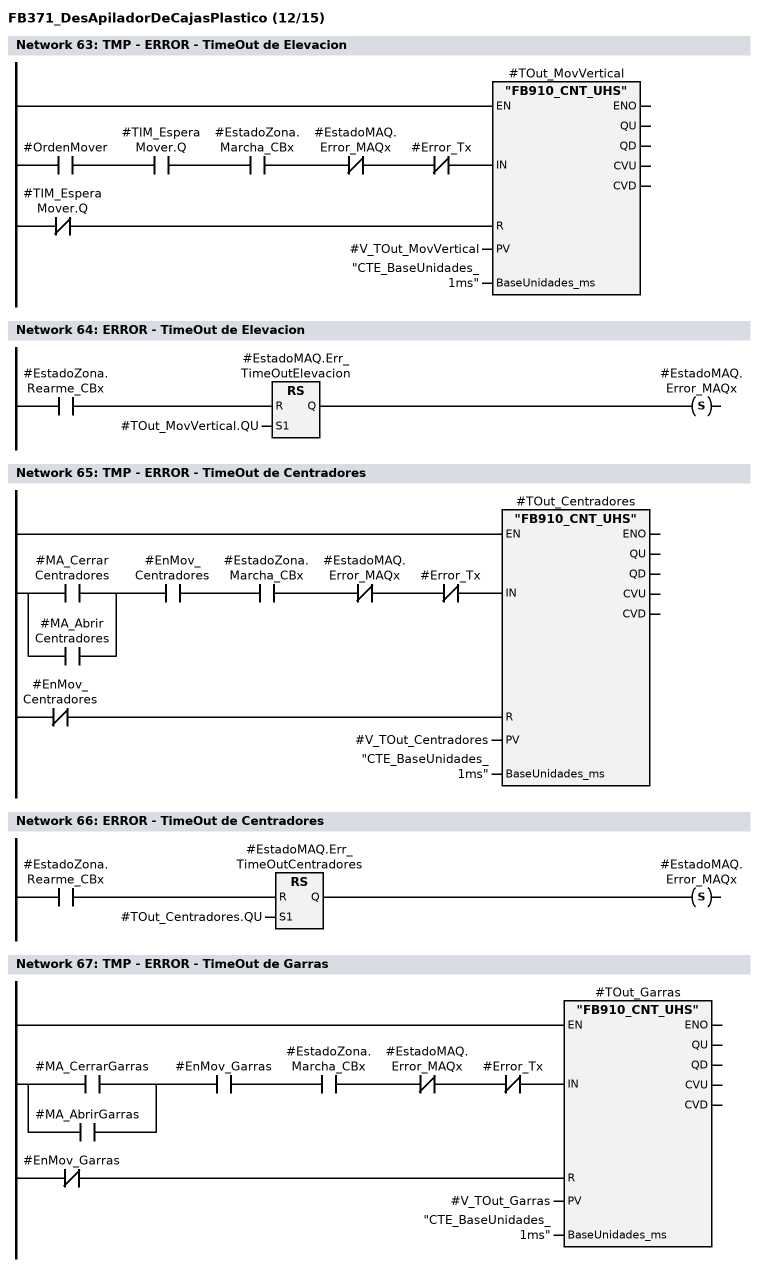
   RUNG wire#powerrail
      #TOut_MovVertical(IN := wire#w1, R := wire#w2, PV := #V_TOut_MovVertical, BaseUnidades_ms := "CTE_BaseUnidades_1ms", QU =>, QD =>, CVU =>, CVD =>)
   END_RUNG
   RUNG wire#powerrail
      Contact( #OrdenMover )
      Contact( #TIM_EsperaMover.Q )
      Contact( #EstadoZona.Marcha_CBx )
      I_Contact( #EstadoMAQ.Error_MAQx )
      I_Contact( #Error_Tx )
   END_RUNG wire#w1
   RUNG wire#powerrail
      I_Contact( #TIM_EsperaMover.Q )
   END_RUNG wire#w2
   // the same network as SCL:
   #TOut_MovVertical(IN := #OrdenMover AND #TIM_EsperaMover.Q AND #EstadoZona.Marcha_CBx AND NOT #EstadoMAQ.Error_MAQx AND NOT #Error_Tx,   // "FB910_CNT_UHS"
                     R := NOT #TIM_EsperaMover.Q,
                     PV := #V_TOut_MovVertical,
                     BaseUnidades_ms := "CTE_BaseUnidades_1ms");
END_REGION

REGION Network 64: ERROR - TimeOut de Elevacion
   RUNG wire#powerrail
      Contact( #EstadoZona.Rearme_CBx )
      S_RS(operand := #EstadoMAQ.Err_TimeOutElevacion, s1 := #TOut_MovVertical.QU)
      S_Coil( #EstadoMAQ.Error_MAQx )
   END_RUNG
   // the same network as SCL:
   IF #EstadoZona.Rearme_CBx THEN
       #EstadoMAQ.Err_TimeOutElevacion := FALSE;   // RS flip-flop
   END_IF;
   IF #TOut_MovVertical.QU THEN #EstadoMAQ.Err_TimeOutElevacion := TRUE; END_IF;
   IF #EstadoMAQ.Err_TimeOutElevacion THEN #EstadoMAQ.Error_MAQx := TRUE; END_IF;
END_REGION

REGION Network 65: TMP - ERROR - TimeOut de Centradores
   RUNG wire#powerrail
      #TOut_Centradores(IN := wire#w2, R := wire#w3, PV := #V_TOut_Centradores, BaseUnidades_ms := "CTE_BaseUnidades_1ms", QU =>, QD =>, CVU =>, CVD =>)
   END_RUNG
   RUNG wire#powerrail
      Contact( #MA_CerrarCentradores )
      wire#w1
      Contact( #EnMov_Centradores )
      Contact( #EstadoZona.Marcha_CBx )
      I_Contact( #EstadoMAQ.Error_MAQx )
      I_Contact( #Error_Tx )
   END_RUNG wire#w2
   RUNG wire#powerrail
      Contact( #MA_AbrirCentradores )
   END_RUNG wire#w1
   RUNG wire#powerrail
      I_Contact( #EnMov_Centradores )
   END_RUNG wire#w3
   // the same network as SCL:
   #TOut_Centradores(IN := (#MA_CerrarCentradores OR #MA_AbrirCentradores) AND #EnMov_Centradores AND #EstadoZona.Marcha_CBx AND NOT #EstadoMAQ.Error_MAQx AND NOT #Error_Tx,   // "FB910_CNT_UHS"
                     R := NOT #EnMov_Centradores,
                     PV := #V_TOut_Centradores,
                     BaseUnidades_ms := "CTE_BaseUnidades_1ms");
END_REGION

REGION Network 66: ERROR - TimeOut de Centradores
   RUNG wire#powerrail
      Contact( #EstadoZona.Rearme_CBx )
      S_RS(operand := #EstadoMAQ.Err_TimeOutCentradores, s1 := #TOut_Centradores.QU)
      S_Coil( #EstadoMAQ.Error_MAQx )
   END_RUNG
   // the same network as SCL:
   IF #EstadoZona.Rearme_CBx THEN
       #EstadoMAQ.Err_TimeOutCentradores := FALSE;   // RS flip-flop
   END_IF;
   IF #TOut_Centradores.QU THEN #EstadoMAQ.Err_TimeOutCentradores := TRUE; END_IF;
   IF #EstadoMAQ.Err_TimeOutCentradores THEN #EstadoMAQ.Error_MAQx := TRUE; END_IF;
END_REGION

REGION Network 67: TMP - ERROR - TimeOut de Garras
   RUNG wire#powerrail
      #TOut_Garras(IN := wire#w2, R := wire#w3, PV := #V_TOut_Garras, BaseUnidades_ms := "CTE_BaseUnidades_1ms", QU =>, QD =>, CVU =>, CVD =>)
   END_RUNG
   RUNG wire#powerrail
      Contact( #MA_CerrarGarras )
      wire#w1
      Contact( #EnMov_Garras )
      Contact( #EstadoZona.Marcha_CBx )
      I_Contact( #EstadoMAQ.Error_MAQx )
      I_Contact( #Error_Tx )
   END_RUNG wire#w2
   RUNG wire#powerrail
      Contact( #MA_AbrirGarras )
   END_RUNG wire#w1
   RUNG wire#powerrail
      I_Contact( #EnMov_Garras )
   END_RUNG wire#w3
   // the same network as SCL:
   #TOut_Garras(IN := (#MA_CerrarGarras OR #MA_AbrirGarras) AND #EnMov_Garras AND #EstadoZona.Marcha_CBx AND NOT #EstadoMAQ.Error_MAQx AND NOT #Error_Tx,   // "FB910_CNT_UHS"
                R := NOT #EnMov_Garras,
                PV := #V_TOut_Garras,
                BaseUnidades_ms := "CTE_BaseUnidades_1ms");
END_REGION

REGION Network 68: ERROR - TimeOut de Garras
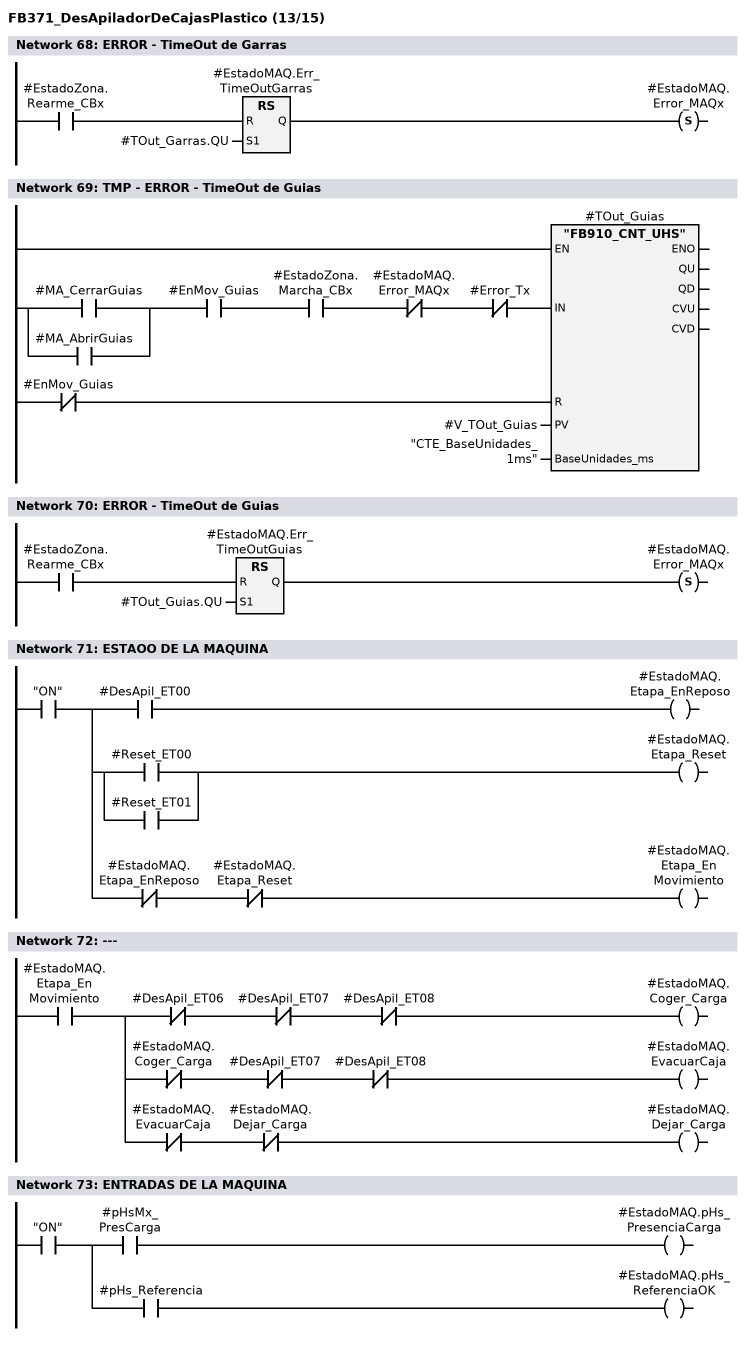
   RUNG wire#powerrail
      Contact( #EstadoZona.Rearme_CBx )
      S_RS(operand := #EstadoMAQ.Err_TimeOutGarras, s1 := #TOut_Garras.QU)
      S_Coil( #EstadoMAQ.Error_MAQx )
   END_RUNG
   // the same network as SCL:
   IF #EstadoZona.Rearme_CBx THEN
       #EstadoMAQ.Err_TimeOutGarras := FALSE;   // RS flip-flop
   END_IF;
   IF #TOut_Garras.QU THEN #EstadoMAQ.Err_TimeOutGarras := TRUE; END_IF;
   IF #EstadoMAQ.Err_TimeOutGarras THEN #EstadoMAQ.Error_MAQx := TRUE; END_IF;
END_REGION

REGION Network 69: TMP - ERROR - TimeOut de Guias
   RUNG wire#powerrail
      #TOut_Guias(IN := wire#w2, R := wire#w3, PV := #V_TOut_Guias, BaseUnidades_ms := "CTE_BaseUnidades_1ms", QU =>, QD =>, CVU =>, CVD =>)
   END_RUNG
   RUNG wire#powerrail
      Contact( #MA_CerrarGuias )
      wire#w1
      Contact( #EnMov_Guias )
      Contact( #EstadoZona.Marcha_CBx )
      I_Contact( #EstadoMAQ.Error_MAQx )
      I_Contact( #Error_Tx )
   END_RUNG wire#w2
   RUNG wire#powerrail
      Contact( #MA_AbrirGuias )
   END_RUNG wire#w1
   RUNG wire#powerrail
      I_Contact( #EnMov_Guias )
   END_RUNG wire#w3
   // the same network as SCL:
   #TOut_Guias(IN := (#MA_CerrarGuias OR #MA_AbrirGuias) AND #EnMov_Guias AND #EstadoZona.Marcha_CBx AND NOT #EstadoMAQ.Error_MAQx AND NOT #Error_Tx,   // "FB910_CNT_UHS"
               R := NOT #EnMov_Guias,
               PV := #V_TOut_Guias,
               BaseUnidades_ms := "CTE_BaseUnidades_1ms");
END_REGION

REGION Network 70: ERROR - TimeOut de Guias
   RUNG wire#powerrail
      Contact( #EstadoZona.Rearme_CBx )
      S_RS(operand := #EstadoMAQ.Err_TimeOutGuias, s1 := #TOut_Guias.QU)
      S_Coil( #EstadoMAQ.Error_MAQx )
   END_RUNG
   // the same network as SCL:
   IF #EstadoZona.Rearme_CBx THEN
       #EstadoMAQ.Err_TimeOutGuias := FALSE;   // RS flip-flop
   END_IF;
   IF #TOut_Guias.QU THEN #EstadoMAQ.Err_TimeOutGuias := TRUE; END_IF;
   IF #EstadoMAQ.Err_TimeOutGuias THEN #EstadoMAQ.Error_MAQx := TRUE; END_IF;
END_REGION

REGION Network 71: ESTAOO DE LA MAQUINA
   RUNG wire#powerrail
      Contact( "ON" )
      wire#w1
      Contact( #DesApil_ET00 )
      Coil( #EstadoMAQ.Etapa_EnReposo )
   END_RUNG
   RUNG wire#w1
      Contact( #Reset_ET00 )
      wire#w2
      Coil( #EstadoMAQ.Etapa_Reset )
   END_RUNG
   RUNG wire#w1
      Contact( #Reset_ET01 )
   END_RUNG wire#w2
   RUNG wire#w1
      I_Contact( #EstadoMAQ.Etapa_EnReposo )
      I_Contact( #EstadoMAQ.Etapa_Reset )
      Coil( #EstadoMAQ.Etapa_EnMovimiento )
   END_RUNG
   // the same network as SCL:
   #EstadoMAQ.Etapa_EnReposo := "ON" AND #DesApil_ET00;
   #EstadoMAQ.Etapa_Reset := "ON" AND (#Reset_ET00 OR #Reset_ET01);
   #EstadoMAQ.Etapa_EnMovimiento := "ON" AND NOT #EstadoMAQ.Etapa_EnReposo AND NOT #EstadoMAQ.Etapa_Reset;
END_REGION

REGION Network 72: ---
   RUNG wire#powerrail
      Contact( #EstadoMAQ.Etapa_EnMovimiento )
      wire#w1
      I_Contact( #DesApil_ET06 )
      I_Contact( #DesApil_ET07 )
      I_Contact( #DesApil_ET08 )
      Coil( #EstadoMAQ.Coger_Carga )
   END_RUNG
   RUNG wire#w1
      I_Contact( #EstadoMAQ.Coger_Carga )
      I_Contact( #DesApil_ET07 )
      I_Contact( #DesApil_ET08 )
      Coil( #EstadoMAQ.EvacuarCaja )
   END_RUNG
   RUNG wire#w1
      I_Contact( #EstadoMAQ.EvacuarCaja )
      I_Contact( #EstadoMAQ.Dejar_Carga )
      Coil( #EstadoMAQ.Dejar_Carga )
   END_RUNG
   // the same network as SCL:
   #EstadoMAQ.Coger_Carga := #EstadoMAQ.Etapa_EnMovimiento AND NOT #DesApil_ET06 AND NOT #DesApil_ET07 AND NOT #DesApil_ET08;
   #EstadoMAQ.EvacuarCaja := #EstadoMAQ.Etapa_EnMovimiento AND NOT #EstadoMAQ.Coger_Carga AND NOT #DesApil_ET07 AND NOT #DesApil_ET08;
   #EstadoMAQ.Dejar_Carga := #EstadoMAQ.Etapa_EnMovimiento AND NOT #EstadoMAQ.EvacuarCaja AND NOT #EstadoMAQ.Dejar_Carga;
END_REGION

REGION Network 73: ENTRADAS DE LA MAQUINA
   RUNG wire#powerrail
      Contact( "ON" )
      wire#w1
      Contact( #pHsMx_PresCarga )
      Coil( #EstadoMAQ.pHs_PresenciaCarga )
   END_RUNG
   RUNG wire#w1
      Contact( #pHs_Referencia )
      Coil( #EstadoMAQ.pHs_ReferenciaOK )
   END_RUNG
   // the same network as SCL:
   #EstadoMAQ.pHs_PresenciaCarga := "ON" AND #pHsMx_PresCarga;
   #EstadoMAQ.pHs_ReferenciaOK := "ON" AND #pHs_Referencia;
END_REGION

REGION Network 74: ---
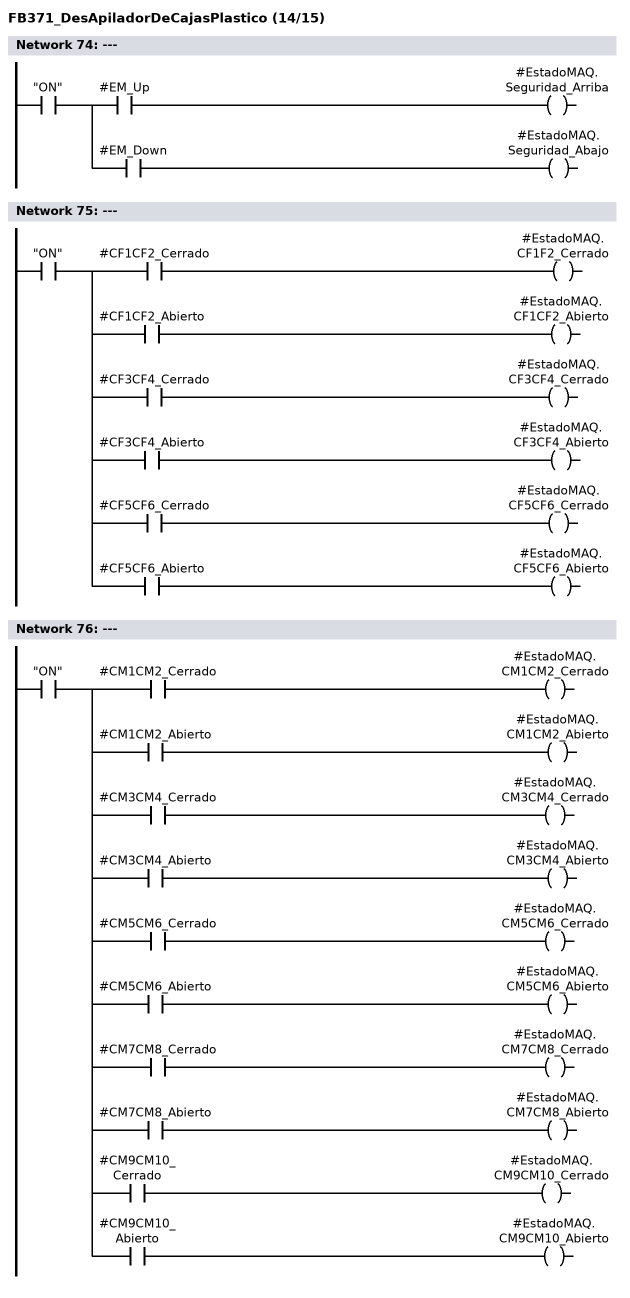
   RUNG wire#powerrail
      Contact( "ON" )
      wire#w1
      Contact( #EM_Up )
      Coil( #EstadoMAQ.Seguridad_Arriba )
   END_RUNG
   RUNG wire#w1
      Contact( #EM_Down )
      Coil( #EstadoMAQ.Seguridad_Abajo )
   END_RUNG
   // the same network as SCL:
   #EstadoMAQ.Seguridad_Arriba := "ON" AND #EM_Up;
   #EstadoMAQ.Seguridad_Abajo := "ON" AND #EM_Down;
END_REGION

REGION Network 75: ---
   RUNG wire#powerrail
      Contact( "ON" )
      wire#w1
      Contact( #CF1CF2_Cerrado )
      Coil( #EstadoMAQ.CF1F2_Cerrado )
   END_RUNG
   RUNG wire#w1
      Contact( #CF1CF2_Abierto )
      Coil( #EstadoMAQ.CF1CF2_Abierto )
   END_RUNG
   RUNG wire#w1
      Contact( #CF3CF4_Cerrado )
      Coil( #EstadoMAQ.CF3CF4_Cerrado )
   END_RUNG
   RUNG wire#w1
      Contact( #CF3CF4_Abierto )
      Coil( #EstadoMAQ.CF3CF4_Abierto )
   END_RUNG
   RUNG wire#w1
      Contact( #CF5CF6_Cerrado )
      Coil( #EstadoMAQ.CF5CF6_Cerrado )
   END_RUNG
   RUNG wire#w1
      Contact( #CF5CF6_Abierto )
      Coil( #EstadoMAQ.CF5CF6_Abierto )
   END_RUNG
   // the same network as SCL:
   #EstadoMAQ.CF1F2_Cerrado := "ON" AND #CF1CF2_Cerrado;
   #EstadoMAQ.CF1CF2_Abierto := "ON" AND #CF1CF2_Abierto;
   #EstadoMAQ.CF3CF4_Cerrado := "ON" AND #CF3CF4_Cerrado;
   #EstadoMAQ.CF3CF4_Abierto := "ON" AND #CF3CF4_Abierto;
   #EstadoMAQ.CF5CF6_Cerrado := "ON" AND #CF5CF6_Cerrado;
   #EstadoMAQ.CF5CF6_Abierto := "ON" AND #CF5CF6_Abierto;
END_REGION

REGION Network 76: ---
   RUNG wire#powerrail
      Contact( "ON" )
      wire#w1
      Contact( #CM1CM2_Cerrado )
      Coil( #EstadoMAQ.CM1CM2_Cerrado )
   END_RUNG
   RUNG wire#w1
      Contact( #CM1CM2_Abierto )
      Coil( #EstadoMAQ.CM1CM2_Abierto )
   END_RUNG
   RUNG wire#w1
      Contact( #CM3CM4_Cerrado )
      Coil( #EstadoMAQ.CM3CM4_Cerrado )
   END_RUNG
   RUNG wire#w1
      Contact( #CM3CM4_Abierto )
      Coil( #EstadoMAQ.CM3CM4_Abierto )
   END_RUNG
   RUNG wire#w1
      Contact( #CM5CM6_Cerrado )
      Coil( #EstadoMAQ.CM5CM6_Cerrado )
   END_RUNG
   RUNG wire#w1
      Contact( #CM5CM6_Abierto )
      Coil( #EstadoMAQ.CM5CM6_Abierto )
   END_RUNG
   RUNG wire#w1
      Contact( #CM7CM8_Cerrado )
      Coil( #EstadoMAQ.CM7CM8_Cerrado )
   END_RUNG
   RUNG wire#w1
      Contact( #CM7CM8_Abierto )
      Coil( #EstadoMAQ.CM7CM8_Abierto )
   END_RUNG
   RUNG wire#w1
      Contact( #CM9CM10_Cerrado )
      Coil( #EstadoMAQ.CM9CM10_Cerrado )
   END_RUNG
   RUNG wire#w1
      Contact( #CM9CM10_Abierto )
      Coil( #EstadoMAQ.CM9CM10_Abierto )
   END_RUNG
   // the same network as SCL:
   #EstadoMAQ.CM1CM2_Cerrado := "ON" AND #CM1CM2_Cerrado;
   #EstadoMAQ.CM1CM2_Abierto := "ON" AND #CM1CM2_Abierto;
   #EstadoMAQ.CM3CM4_Cerrado := "ON" AND #CM3CM4_Cerrado;
   #EstadoMAQ.CM3CM4_Abierto := "ON" AND #CM3CM4_Abierto;
   #EstadoMAQ.CM5CM6_Cerrado := "ON" AND #CM5CM6_Cerrado;
   #EstadoMAQ.CM5CM6_Abierto := "ON" AND #CM5CM6_Abierto;
   #EstadoMAQ.CM7CM8_Cerrado := "ON" AND #CM7CM8_Cerrado;
   #EstadoMAQ.CM7CM8_Abierto := "ON" AND #CM7CM8_Abierto;
   #EstadoMAQ.CM9CM10_Cerrado := "ON" AND #CM9CM10_Cerrado;
   #EstadoMAQ.CM9CM10_Abierto := "ON" AND #CM9CM10_Abierto;
END_REGION

REGION Network 77: ---
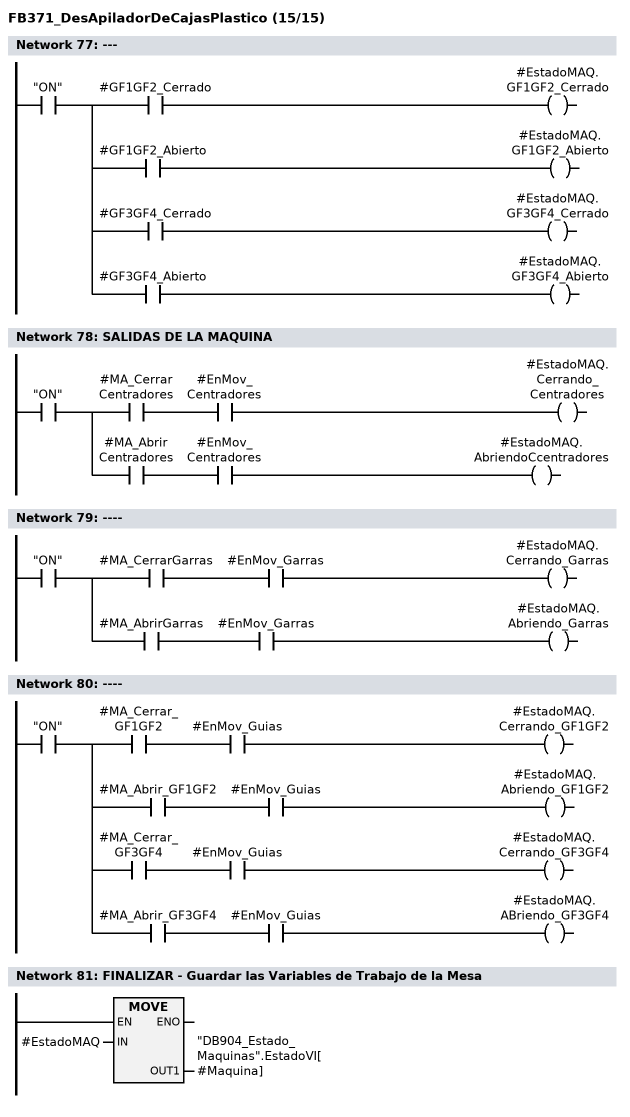
   RUNG wire#powerrail
      Contact( "ON" )
      wire#w1
      Contact( #GF1GF2_Cerrado )
      Coil( #EstadoMAQ.GF1GF2_Cerrado )
   END_RUNG
   RUNG wire#w1
      Contact( #GF1GF2_Abierto )
      Coil( #EstadoMAQ.GF1GF2_Abierto )
   END_RUNG
   RUNG wire#w1
      Contact( #GF3GF4_Cerrado )
      Coil( #EstadoMAQ.GF3GF4_Cerrado )
   END_RUNG
   RUNG wire#w1
      Contact( #GF3GF4_Abierto )
      Coil( #EstadoMAQ.GF3GF4_Abierto )
   END_RUNG
   // the same network as SCL:
   #EstadoMAQ.GF1GF2_Cerrado := "ON" AND #GF1GF2_Cerrado;
   #EstadoMAQ.GF1GF2_Abierto := "ON" AND #GF1GF2_Abierto;
   #EstadoMAQ.GF3GF4_Cerrado := "ON" AND #GF3GF4_Cerrado;
   #EstadoMAQ.GF3GF4_Abierto := "ON" AND #GF3GF4_Abierto;
END_REGION

REGION Network 78: SALIDAS DE LA MAQUINA
   RUNG wire#powerrail
      Contact( "ON" )
      wire#w1
      Contact( #MA_CerrarCentradores )
      Contact( #EnMov_Centradores )
      Coil( #EstadoMAQ.Cerrando_Centradores )
   END_RUNG
   RUNG wire#w1
      Contact( #MA_AbrirCentradores )
      Contact( #EnMov_Centradores )
      Coil( #EstadoMAQ.AbriendoCcentradores )
   END_RUNG
   // the same network as SCL:
   #EstadoMAQ.Cerrando_Centradores := "ON" AND #MA_CerrarCentradores AND #EnMov_Centradores;
   #EstadoMAQ.AbriendoCcentradores := "ON" AND #MA_AbrirCentradores AND #EnMov_Centradores;
END_REGION

REGION Network 79: ----
   RUNG wire#powerrail
      Contact( "ON" )
      wire#w1
      Contact( #MA_CerrarGarras )
      Contact( #EnMov_Garras )
      Coil( #EstadoMAQ.Cerrando_Garras )
   END_RUNG
   RUNG wire#w1
      Contact( #MA_AbrirGarras )
      Contact( #EnMov_Garras )
      Coil( #EstadoMAQ.Abriendo_Garras )
   END_RUNG
   // the same network as SCL:
   #EstadoMAQ.Cerrando_Garras := "ON" AND #MA_CerrarGarras AND #EnMov_Garras;
   #EstadoMAQ.Abriendo_Garras := "ON" AND #MA_AbrirGarras AND #EnMov_Garras;
END_REGION

REGION Network 80: ----
   RUNG wire#powerrail
      Contact( "ON" )
      wire#w1
      Contact( #MA_Cerrar_GF1GF2 )
      Contact( #EnMov_Guias )
      Coil( #EstadoMAQ.Cerrando_GF1GF2 )
   END_RUNG
   RUNG wire#w1
      Contact( #MA_Abrir_GF1GF2 )
      Contact( #EnMov_Guias )
      Coil( #EstadoMAQ.Abriendo_GF1GF2 )
   END_RUNG
   RUNG wire#w1
      Contact( #MA_Cerrar_GF3GF4 )
      Contact( #EnMov_Guias )
      Coil( #EstadoMAQ.Cerrando_GF3GF4 )
   END_RUNG
   RUNG wire#w1
      Contact( #MA_Abrir_GF3GF4 )
      Contact( #EnMov_Guias )
      Coil( #EstadoMAQ.ABriendo_GF3GF4 )
   END_RUNG
   // the same network as SCL:
   #EstadoMAQ.Cerrando_GF1GF2 := "ON" AND #MA_Cerrar_GF1GF2 AND #EnMov_Guias;
   #EstadoMAQ.Abriendo_GF1GF2 := "ON" AND #MA_Abrir_GF1GF2 AND #EnMov_Guias;
   #EstadoMAQ.Cerrando_GF3GF4 := "ON" AND #MA_Cerrar_GF3GF4 AND #EnMov_Guias;
   #EstadoMAQ.ABriendo_GF3GF4 := "ON" AND #MA_Abrir_GF3GF4 AND #EnMov_Guias;
END_REGION

REGION Network 81: FINALIZAR - Guardar las Variables de Trabajo de la Mesa
   RUNG wire#powerrail
      Move(in := #EstadoMAQ, out1 => "DB904_Estado_Maquinas".EstadoVI[#Maquina])
   END_RUNG
   // the same network as SCL:
   "DB904_Estado_Maquinas".EstadoVI[#Maquina] := #EstadoMAQ;
END_REGION
END_FUNCTION_BLOCK
